// TwinCAT 3 PLC project ED_PROG
// ProgramVersion: 3.1.4026.12
// libraries:
//   Tc2_OpcUA, * (Beckhoff Automation GmbH)
//   Tc2_Standard, * (Beckhoff Automation GmbH)
//   Tc2_System, * (Beckhoff Automation GmbH)
//   Tc2_Utilities, * (Beckhoff Automation GmbH)
//   Tc3_Module, * (Beckhoff Automation GmbH)
// project tree:
//   GVLs/ opc.TcGVL, plccomms.TcGVL
//   / PlcTask.TcTTO
//   POUs/ alarm_manager.TcPOU, idle.TcPOU, cip.TcPOU, example_loop_control.TcPOU, faults.TcPOU, interlocks.TcPOU, io_mapping.TcPOU, communications.TcPOU (not stored), general.TcPOU, manual_mode.TcPOU, maint_mode.TcPOU, opc_control.TcPOU (not stored), opc_mapping.TcPOU, output_mapping.TcPOU, pump_manager.TcPOU, state_transition.TcPOU (not stored), stopping_mode.TcPOU, valve_manager.TcPOU
//   POUs/Function Blocks/ ramp.TcPOU, alarm.TcPOU, analog_scaling.TcPOU (not stored), date_time.TcPOU (not stored), motor_starter.TcPOU (not stored), motor_vfd.TcPOU (not stored), valve_analog.TcPOU (not stored), valve_digital.TcPOU (not stored)
// real-time tasks:
//   TASK PlcTask: cycle T#10ms, priority 20, ADS port 350
//   TASK twinsafe: cycle T#10ms, priority 1, ADS port 301
// I/O:
//   DEVICE Device 1 (EtherCAT), AmsNetId 10.60.1.103.2.1
//     Term 1 (EK1200) [EK1200-5000 EtherCAT Power supply (2A E-Bus)]
//       Term 2 (EL3058) [EL3058 8Ch. Ana. Input 4-20mA]
//       Term 3 (EL3058) [EL3058 8Ch. Ana. Input 4-20mA]
//       Term 4 (EL4124) [EL4124 4Ch. Ana. Output 4-20mA, 16bit]
//       Term 5 (EL4124) [EL4124 4Ch. Ana. Output 4-20mA, 16bit]
//       Term 6 (EL4124) [EL4124 4Ch. Ana. Output 4-20mA, 16bit]
//       Term 7 (EL1859) [EL1859 8Ch. Dig. Input 24V, 3ms, 8Ch. Dig. Output 24V, 0.5A]
//       Term 8 (EL1859) [EL1859 8Ch. Dig. Input 24V, 3ms, 8Ch. Dig. Output 24V, 0.5A]
//       Term 9 (EL1859) [EL1859 8Ch. Dig. Input 24V, 3ms, 8Ch. Dig. Output 24V, 0.5A]
//       Term 10 (EL1904) [EL1904, 4 Ch. Safety Input 24V, TwinSAFE]
//         modules: Module 1 (FSOES)
//       Term 11 (EL2911) [EL2911, Potential supply terminal (10 A) with 4 Ch. Safety Inputs, TwinSAFE]
//         modules: Module 2 (FSOUT), Module 3 (DEVICEIO), Module 4 (FSLOGIC)
//       Term 12 (EK1110) [EK1110 EtherCAT extension]
//     Term 20 (EK1100-0018) [EK1100-0018 EtherCAT-Koppler (2A E-Bus, erw. Surge Schutz)]
//       Term 21 (EL3058) [EL3058 8Ch. Ana. Input 4-20mA]
//       Term 22 (EL3058) [EL3058 8Ch. Ana. Input 4-20mA]
//       Term 23 (EL3058) [EL3058 8Ch. Ana. Input 4-20mA]
//       Term 24 (EL3058) [EL3058 8Ch. Ana. Input 4-20mA]
//       Term 25 (EL3058) [EL3058 8Ch. Ana. Input 4-20mA]
//       Term 26 (EL4124) [EL4124 4Ch. Ana. Output 4-20mA, 16bit]
//       Term 27 (EL4124) [EL4124 4Ch. Ana. Output 4-20mA, 16bit]
//       Term 28 (EL1859) [EL1859 8Ch. Dig. Input 24V, 3ms, 8Ch. Dig. Output 24V, 0.5A]
//       Term 29 (EL1859) [EL1859 8Ch. Dig. Input 24V, 3ms, 8Ch. Dig. Output 24V, 0.5A]
//       Term 30 (EL9011) [EL9011 End Terminal]
//     Term 31 (EK1914) [EK1914, 2 Ch. Safety Input/Output 24V,  TwinSAFE]
//       modules: Module 1 (FSOE), Module 2 (DIO)
//       Term 32 (EL1859) [EL1859 8Ch. Dig. Input 24V, 3ms, 8Ch. Dig. Output 24V, 0.5A]
//       Term 33 (EL1859) [EL1859 8Ch. Dig. Input 24V, 3ms, 8Ch. Dig. Output 24V, 0.5A]
//       Term 34 (EL1904) [EL1904, 4 Ch. Safety Input 24V, TwinSAFE]
//         modules: Module 1 (FSOES)
//       Term 35 (EL9011) [EL9011 End Terminal]
//   DEVICE Device 4 (EtherCAT), AmsNetId 10.60.1.103.5.1
//     Term 13 (EK1100-0018) [EK1100-0018 EtherCAT-Koppler (2A E-Bus, erw. Surge Schutz)]
//       Term 14 (EL3058) [EL3058 8Ch. Ana. Input 4-20mA]
//       Term 15 (EL3058) [EL3058 8Ch. Ana. Input 4-20mA]
//       Term 16 (EL3058) [EL3058 8Ch. Ana. Input 4-20mA]
//       Term 17 (EL3058) [EL3058 8Ch. Ana. Input 4-20mA]
//       Term 18 (EL3058) [EL3058 8Ch. Ana. Input 4-20mA]
//       Term 19 (EL4124) [EL4124 4Ch. Ana. Output 4-20mA, 16bit]
//       Term 20 (EL4124) [EL4124 4Ch. Ana. Output 4-20mA, 16bit]
//       Term 21 (EL1859) [EL1859 8Ch. Dig. Input 24V, 3ms, 8Ch. Dig. Output 24V, 0.5A]
//       Term 22 (EL1859) [EL1859 8Ch. Dig. Input 24V, 3ms, 8Ch. Dig. Output 24V, 0.5A]
//       Term 41 (EL9011) [EL9011 End Terminal]
//     Term 31 (EK1914) [EK1914, 2 Ch. Safety Input/Output 24V,  TwinSAFE]
//       modules: Module 1 (FSOE), Module 2 (DIO)
//       Term 32 (EL1859) [EL1859 8Ch. Dig. Input 24V, 3ms, 8Ch. Dig. Output 24V, 0.5A]
//       Term 33 (EL1859) [EL1859 8Ch. Dig. Input 24V, 3ms, 8Ch. Dig. Output 24V, 0.5A]
//       Term 34 (EL1904) [EL1904, 4 Ch. Safety Input 24V, TwinSAFE]
//         modules: Module 1 (FSOES)
//       Term 42 (EL9011) [EL9011 End Terminal]
//     Term 40 (EK1100) [EK1100 EtherCAT Coupler (2A E-Bus)]
//       Term 41 (EL3058) [EL3058 8Ch. Ana. Input 4-20mA]
//       Term 42 (EL4124) [EL4124 4Ch. Ana. Output 4-20mA, 16bit]
//       Term 43 (EL1859) [EL1859 8Ch. Dig. Input 24V, 3ms, 8Ch. Dig. Output 24V, 0.5A]
//       Term 44 (EL2911) [EL2911, Potential supply terminal (10 A) with 4 Ch. Safety Inputs, TwinSAFE]
//         modules: Module 1 (FSOE), Module 2 (FSOUT), Module 3 (DEVICEIO), Module 4 (FSLOGIC)
//       Term 43 (EL9011) [EL9011 End Terminal]
// variable links:
//   Device 1 (EtherCAT) <-> Device 1 (EtherCAT)/Term 1 (EK1200)/Term 11 (EL2911)
//     Term 31 (EK1914)/Module 1 (FSOE)/Inputs/FSOE <-> ConnectionOutputs/Message_18 RxPDO
//     Term 31 (EK1914)/Module 1 (FSOE)/Outputs/FSOE <-> ConnectionInputs/Message_18 TxPDO
//   ED2_PROG Instance <-> Device 1 (EtherCAT)/Term 1 (EK1200)/Term 2 (EL3058)
//     PlcTask Inputs/io_mapping.u_3112_b_speed_feedback_raw_input <-> AI Standard Channel 1/Value
//     PlcTask Inputs/io_mapping.u_3160_b_speed_feedback_raw_input <-> AI Standard Channel 4/Value
//     PlcTask Inputs/io_mapping.u_3212_b_speed_feedback_raw_input <-> AI Standard Channel 2/Value
//     PlcTask Inputs/io_mapping.u_3260_b_speed_feedback_raw_input <-> AI Standard Channel 5/Value
//     PlcTask Inputs/io_mapping.u_3312_b_speed_feedback_raw_input <-> AI Standard Channel 3/Value
//     PlcTask Inputs/io_mapping.u_3360_b_speed_feedback_raw_input <-> AI Standard Channel 6/Value
//     PlcTask Inputs/io_mapping.u_3370_b_speed_feedback_raw_input <-> AI Standard Channel 7/Value
//   ED2_PROG Instance <-> Device 1 (EtherCAT)/Term 1 (EK1200)/Term 4 (EL4124)
//     PlcTask Outputs/output_mapping.u_3112_b_speed_command_io <-> AO Output Channel 1/Analog output
//     PlcTask Outputs/output_mapping.u_3160_b_speed_command_io <-> AO Output Channel 4/Analog output
//     PlcTask Outputs/output_mapping.u_3212_b_speed_command_io <-> AO Output Channel 2/Analog output
//     PlcTask Outputs/output_mapping.u_3312_b_speed_command_io <-> AO Output Channel 3/Analog output
//   ED2_PROG Instance <-> Device 1 (EtherCAT)/Term 1 (EK1200)/Term 5 (EL4124)
//     PlcTask Outputs/output_mapping.u_3260_b_speed_command_io <-> AO Output Channel 1/Analog output
//     PlcTask Outputs/output_mapping.u_3360_b_speed_command_io <-> AO Output Channel 2/Analog output
//     PlcTask Outputs/output_mapping.u_3370_b_speed_command_io <-> AO Output Channel 3/Analog output
//   ED2_PROG Instance <-> Device 1 (EtherCAT)/Term 1 (EK1200)/Term 7 (EL1859)
//     PlcTask Inputs/io_mapping.u_3112_b_fault_feedback <-> Channel 1/Input
//     PlcTask Inputs/io_mapping.u_3160_b_fault_feedback <-> Channel 7/Input
//     PlcTask Inputs/io_mapping.u_3212_b_fault_feedback <-> Channel 3/Input
//     PlcTask Inputs/io_mapping.u_3312_b_fault_feedback <-> Channel 5/Input
//     PlcTask Inputs/io_mapping.u_3112_b_run_feedback <-> Channel 2/Input
//     PlcTask Inputs/io_mapping.u_3160_b_run_feedback <-> Channel 8/Input
//     PlcTask Inputs/io_mapping.u_3212_b_run_feedback <-> Channel 4/Input
//     PlcTask Inputs/io_mapping.u_3312_b_run_feedback <-> Channel 6/Input
//     PlcTask Outputs/output_mapping.u_3112_b_fault_reset_io <-> Channel 10/Output
//     PlcTask Outputs/output_mapping.u_3160_b_fault_reset_io <-> Channel 16/Output
//     PlcTask Outputs/output_mapping.u_3212_b_fault_reset_io <-> Channel 12/Output
//     PlcTask Outputs/output_mapping.u_3312_b_fault_reset_io <-> Channel 14/Output
//     PlcTask Outputs/output_mapping.u_3112_b_run_command_io <-> Channel 9/Output
//     PlcTask Outputs/output_mapping.u_3160_b_run_command_io <-> Channel 15/Output
//     PlcTask Outputs/output_mapping.u_3212_b_run_command_io <-> Channel 11/Output
//     PlcTask Outputs/output_mapping.u_3312_b_run_command_io <-> Channel 13/Output
//   ED2_PROG Instance <-> Device 1 (EtherCAT)/Term 1 (EK1200)/Term 8 (EL1859)
//     PlcTask Inputs/io_mapping.u_3260_b_fault_feedback <-> Channel 1/Input
//     PlcTask Inputs/io_mapping.u_3360_b_fault_feedback <-> Channel 3/Input
//     PlcTask Inputs/io_mapping.u_3370_b_fault_feedback <-> Channel 5/Input
//     PlcTask Inputs/io_mapping.u_3260_b_run_feedback <-> Channel 2/Input
//     PlcTask Inputs/io_mapping.u_3360_b_run_feedback <-> Channel 4/Input
//     PlcTask Inputs/io_mapping.u_3370_b_run_feedback <-> Channel 6/Input
//     PlcTask Outputs/output_mapping.u_3260_b_fault_reset_io <-> Channel 10/Output
//     PlcTask Outputs/output_mapping.u_3360_b_fault_reset_io <-> Channel 12/Output
//     PlcTask Outputs/output_mapping.u_3370_b_fault_reset_io <-> Channel 14/Output
//     PlcTask Outputs/output_mapping.u_3260_b_run_command_io <-> Channel 9/Output
//     PlcTask Outputs/output_mapping.u_3360_b_run_command_io <-> Channel 11/Output
//     PlcTask Outputs/output_mapping.u_3370_b_run_command_io <-> Channel 13/Output
//   ED2_PROG Instance <-> Device 1 (EtherCAT)/Term 20 (EK1100-0018)/Term 21 (EL3058)
//     PlcTask Inputs/io_mapping.pt_3119_b_raw_input <-> AI Standard Channel 1/Value
//     PlcTask Inputs/io_mapping.pt_3141_b_raw_input <-> AI Standard Channel 4/Value
//     PlcTask Inputs/io_mapping.pt_3219_b_raw_input <-> AI Standard Channel 2/Value
//     PlcTask Inputs/io_mapping.pt_3241_b_raw_input <-> AI Standard Channel 5/Value
//     PlcTask Inputs/io_mapping.pt_3319_b_raw_input <-> AI Standard Channel 3/Value
//     PlcTask Inputs/io_mapping.pt_3341_b_raw_input <-> AI Standard Channel 6/Value
//     PlcTask Inputs/io_mapping.tt_3118_b_raw_input <-> AI Standard Channel 7/Value
//     PlcTask Inputs/io_mapping.tt_3218_b_raw_input <-> AI Standard Channel 8/Value
//   ED2_PROG Instance <-> Device 1 (EtherCAT)/Term 20 (EK1100-0018)/Term 22 (EL3058)
//     PlcTask Inputs/io_mapping.av_3148_b_position_feedback_raw_input <-> AI Standard Channel 8/Value
//     PlcTask Inputs/io_mapping.tt_3140_b_raw_input <-> AI Standard Channel 2/Value
//     PlcTask Inputs/io_mapping.tt_3240_b_raw_input <-> AI Standard Channel 3/Value
//     PlcTask Inputs/io_mapping.tt_3318_b_raw_input <-> AI Standard Channel 1/Value
//     PlcTask Inputs/io_mapping.tt_3340_b_raw_input <-> AI Standard Channel 4/Value
//   ED2_PROG Instance <-> Device 1 (EtherCAT)/Term 20 (EK1100-0018)/Term 23 (EL3058)
//     PlcTask Inputs/io_mapping.av_3248_b_position_feedback_raw_input <-> AI Standard Channel 1/Value
//     PlcTask Inputs/io_mapping.av_3348_b_position_feedback_raw_input <-> AI Standard Channel 2/Value
//     PlcTask Inputs/io_mapping.lt_3102_b_raw_input <-> AI Standard Channel 3/Value
//     PlcTask Inputs/io_mapping.lt_3153_b_raw_input <-> AI Standard Channel 6/Value
//     PlcTask Inputs/io_mapping.lt_3202_b_raw_input <-> AI Standard Channel 4/Value
//     PlcTask Inputs/io_mapping.lt_3253_b_raw_input <-> AI Standard Channel 7/Value
//     PlcTask Inputs/io_mapping.lt_3302_b_raw_input <-> AI Standard Channel 5/Value
//     PlcTask Inputs/io_mapping.lt_3353_b_raw_input <-> AI Standard Channel 8/Value
//   ED2_PROG Instance <-> Device 1 (EtherCAT)/Term 20 (EK1100-0018)/Term 24 (EL3058)
//     PlcTask Inputs/io_mapping.cct_3120_b_raw_input <-> AI Standard Channel 1/Value
//     PlcTask Inputs/io_mapping.cct_3142_b_raw_input <-> AI Standard Channel 4/Value
//     PlcTask Inputs/io_mapping.cct_3220_b_raw_input <-> AI Standard Channel 2/Value
//     PlcTask Inputs/io_mapping.cct_3242_b_raw_input <-> AI Standard Channel 5/Value
//     PlcTask Inputs/io_mapping.cct_3320_b_raw_input <-> AI Standard Channel 3/Value
//     PlcTask Inputs/io_mapping.cct_3342_b_raw_input <-> AI Standard Channel 6/Value
//   ED2_PROG Instance <-> Device 1 (EtherCAT)/Term 20 (EK1100-0018)/Term 25 (EL3058)
//     PlcTask Inputs/io_mapping.ft_3122_b_raw_input <-> AI Standard Channel 1/Value
//     PlcTask Inputs/io_mapping.ft_3222_b_raw_input <-> AI Standard Channel 2/Value
//     PlcTask Inputs/io_mapping.ft_3322_b_raw_input <-> AI Standard Channel 3/Value
//   ED2_PROG Instance <-> Device 1 (EtherCAT)/Term 20 (EK1100-0018)/Term 26 (EL4124)
//     PlcTask Outputs/output_mapping.av_3148_b_position_command_io <-> AO Output Channel 1/Analog output
//     PlcTask Outputs/output_mapping.av_3248_b_position_command_io <-> AO Output Channel 2/Analog output
//     PlcTask Outputs/output_mapping.av_3348_b_position_command_io <-> AO Output Channel 3/Analog output
//   ED2_PROG Instance <-> Device 1 (EtherCAT)/Term 20 (EK1100-0018)/Term 28 (EL1859)
//     PlcTask Inputs/io_mapping.nv_3135_b_open_feedback <-> Channel 1/Input
//     PlcTask Inputs/io_mapping.nv_3162_b_open_feedback <-> Channel 5/Input
//     PlcTask Inputs/io_mapping.nv_3235_b_open_feedback <-> Channel 2/Input
//     PlcTask Inputs/io_mapping.nv_3335_b_open_feedback <-> Channel 3/Input
//     PlcTask Inputs/io_mapping.nv_3372_b_open_feedback <-> Channel 4/Input
//   ED2_PROG Instance <-> Device 1 (EtherCAT)/Term 20 (EK1100-0018)/Term 29 (EL1859)
//     PlcTask Inputs/io_mapping.nv_3135_b_closed_feedback <-> Channel 1/Input
//     PlcTask Inputs/io_mapping.nv_3162_b_closed_feedback <-> Channel 5/Input
//     PlcTask Inputs/io_mapping.nv_3235_b_closed_feedback <-> Channel 2/Input
//     PlcTask Inputs/io_mapping.nv_3335_b_closed_feedback <-> Channel 3/Input
//     PlcTask Inputs/io_mapping.nv_3372_b_closed_feedback <-> Channel 4/Input
//   ED2_PROG Instance <-> Device 1 (EtherCAT)/Term 31 (EK1914)/Term 32 (EL1859)
//     PlcTask Outputs/output_mapping.nv_3110_b_open_command_io <-> Channel 11/Output
//     PlcTask Outputs/output_mapping.nv_3135_b_open_command_io <-> Channel 12/Output
//     PlcTask Outputs/output_mapping.nv_3162_b_open_command_io <-> Channel 9/Output
//     PlcTask Outputs/output_mapping.nv_3210_b_open_command_io <-> Channel 10/Output
//     PlcTask Outputs/output_mapping.nv_3235_b_open_command_io <-> Channel 14/Output
//     PlcTask Outputs/output_mapping.nv_3310_b_open_command_io <-> Channel 13/Output
//     PlcTask Outputs/output_mapping.nv_3335_b_open_command_io <-> Channel 15/Output
//     PlcTask Outputs/output_mapping.nv_3372_b_open_command_io <-> Channel 16/Output

CONFIGURATION ED_PROG
    RESOURCE PLC ON TwinCAT3
        TASK PlcTask(INTERVAL := T#10ms, PRIORITY := 20);
        PROGRAM communications WITH PlcTask : communications;
        PROGRAM example_loop_control WITH PlcTask : example_loop_control;
        PROGRAM general WITH PlcTask : general;
        PROGRAM interlocks WITH PlcTask : interlocks;
        PROGRAM io_mapping WITH PlcTask : io_mapping;
        PROGRAM opc_control WITH PlcTask : opc_control;
        PROGRAM opc_mapping WITH PlcTask : opc_mapping;
        PROGRAM state_transition WITH PlcTask : state_transition;
        PROGRAM manual_mode WITH PlcTask : manual_mode;
        PROGRAM valve_manager WITH PlcTask : valve_manager;
        PROGRAM stopping_mode WITH PlcTask : stopping_mode;
        PROGRAM pump_manager WITH PlcTask : pump_manager;
        PROGRAM idle WITH PlcTask : idle;
        PROGRAM maint_mode WITH PlcTask : maint_mode;
        PROGRAM faults WITH PlcTask : faults;
        PROGRAM alarm_manager WITH PlcTask : alarm_manager;
        PROGRAM cip WITH PlcTask : cip;
    END_RESOURCE
END_CONFIGURATION

// ---- GVLs/opc.TcGVL
{attribute 'qualified_only'}
{attribute 'global_init_slot' := '50500'}
VAR_GLOBAL PERSISTENT
	//These tags are created here because you cannot write directly to local scoped tags(cpt_3144) from outside the POU
	//They are created here then mapped to the local variables in the POU
	//All tags in this GVL MUST have the {attribute 'OPC.UA.DA' :='1'} string above them in order to be exposed to OPC
	//Tags that are ONLY being read from the HMI have their values set in the opc_mapping program
	
	//------------------------------------------------------------------------------------------------------------------


	//---System date time year-----------------------------------------------------------------------------------------------
	{attribute 'OPC.UA.DA' :='1'}
	popa_0081_system_date_time_year : INT;
	//System date time month
	{attribute 'OPC.UA.DA' :='1'}
	popa_0081_system_date_time_month : INT;
	//System date time day
	{attribute 'OPC.UA.DA' :='1'}
	popa_0081_system_date_time_day : INT;
	//System date time hour
	{attribute 'OPC.UA.DA' :='1'}
	popa_0081_system_date_time_hour : INT;
	//System date time minute
	{attribute 'OPC.UA.DA' :='1'}
	popa_0081_system_date_time_minute : INT;
	//System date time second
	{attribute 'OPC.UA.DA' :='1'}
	popa_0081_system_date_time_second : INT;
	//Hour setpoint for daily reset triggers
	{attribute 'OPC.UA.DA' :='1'}
	popa_0081_daily_reset_hour_setpoint : INT;
	//Minute setpoint for daily reset triggers
	{attribute 'OPC.UA.DA' :='1'}
	popa_0081_daily_reset_minute_setpoint : INT;
	//Alarm acknowledge, acks all alarms, clears lower priority level alarms
	{attribute 'OPC.UA.DA' :='1'}
	popa_0081_alarm_ack : BOOL;
	//Alarm reset, clears higher priority alarms
	{attribute 'OPC.UA.DA' :='1'}
	popa_0081_alarm_reset : BOOL;
	
//----------------------------------------------------------------------------------------------------------------------------------------		
	//State Mode
	{attribute 'OPC.UA.DA' :='1'}
	popa_0081_ed_routine_maint : BOOL;
	{attribute 'OPC.UA.DA' :='1'}
	popa_0081_ed_routine_idle : BOOL;
	{attribute 'OPC.UA.DA' :='1'}
	popa_0081_ed_routine_cip : BOOL;
	{attribute 'OPC.UA.DA' :='1'}
	popa_0081_ed_routine_stop : BOOL;
	{attribute 'OPC.UA.DA' :='1'}
	popa_0081_ed_routine_critical_stop : BOOL;
	
	
	//Safety
	{attribute 'OPC.UA.DA' :='1'}
	popa_0081_ed_safety_reset : BOOL;
	
	
//---HMI Commands--------------------------------------------------------------------------------------------------------------------------------------

	//Setpoints------------------------------------------------------------------------------------------------------------------
	{attribute 'OPC.UA.DA' :='1'}
	popa_0081_idle_pressure_setpoint_request : REAL;
	{attribute 'OPC.UA.DA' :='1'}
	popa_0081_cip_pressure_setpoint_request : REAL;
	{attribute 'OPC.UA.DA' :='1'}
	popa_0081_av_3148_a_hmi_position_request : REAL;
	{attribute 'OPC.UA.DA' :='1'}
	popa_0081_av_3248_a_hmi_position_request : REAL;
	{attribute 'OPC.UA.DA' :='1'}
	popa_0081_av_3348_a_hmi_position_request : REAL;
	
	//Pumps-----------------------------------------------------------------------------------------------------------------------
	{attribute 'OPC.UA.DA' :='1'}
	popa_0081_u_3112_a_hmi_start_request: BOOL;
	{attribute 'OPC.UA.DA' :='1'}
	popa_0081_u_3212_a_hmi_start_request: BOOL;
	{attribute 'OPC.UA.DA' :='1'}
	popa_0081_u_3312_a_hmi_start_request: BOOL;
	{attribute 'OPC.UA.DA' :='1'}
	popa_0081_u_3160_a_hmi_start_request: BOOL;
	{attribute 'OPC.UA.DA' :='1'}
	popa_0081_u_3260_a_hmi_start_request: BOOL;
	{attribute 'OPC.UA.DA' :='1'}
	popa_0081_u_3360_a_hmi_start_request: BOOL;
	{attribute 'OPC.UA.DA' :='1'}
	popa_0081_u_3370_a_hmi_start_request: BOOL;
	{attribute 'OPC.UA.DA' :='1'}
	popa_0091_u_3405_a_hmi_start_request: BOOL;
		
	{attribute 'OPC.UA.DA' :='1'}
	popa_0081_u_3112_a_hmi_speed_request: REAL;
	{attribute 'OPC.UA.DA' :='1'}
	popa_0081_u_3212_a_hmi_speed_request: REAL;
	{attribute 'OPC.UA.DA' :='1'}
	popa_0081_u_3312_a_hmi_speed_request: REAL;
	{attribute 'OPC.UA.DA' :='1'}
	popa_0081_u_3160_a_hmi_speed_request: REAL;
	{attribute 'OPC.UA.DA' :='1'}
	popa_0081_u_3260_a_hmi_speed_request: REAL;
	{attribute 'OPC.UA.DA' :='1'}
	popa_0081_u_3360_a_hmi_speed_request: REAL;
	{attribute 'OPC.UA.DA' :='1'}
	popa_0081_u_3370_a_hmi_speed_request: REAL;
	{attribute 'OPC.UA.DA' :='1'}
	popa_0091_u_3405_a_hmi_speed_request: REAL;
	
	//Valves------------------------------------------------------------------------------------------------------------------------------
	{attribute 'OPC.UA.DA' :='1'}
	popa_0081_nv_3110_a_hmi_open_request: BOOL;
	{attribute 'OPC.UA.DA' :='1'}
	popa_0081_nv_3210_a_hmi_open_request: BOOL;
	{attribute 'OPC.UA.DA' :='1'}
	popa_0081_nv_3310_a_hmi_open_request: BOOL;
	{attribute 'OPC.UA.DA' :='1'}
	popa_0081_nv_3135_a_hmi_open_request: BOOL;
	{attribute 'OPC.UA.DA' :='1'}
	popa_0081_nv_3235_a_hmi_open_request: BOOL;
	{attribute 'OPC.UA.DA' :='1'}
	popa_0081_nv_3335_a_hmi_open_request: BOOL;
	{attribute 'OPC.UA.DA' :='1'}
	popa_0081_nv_3372_a_hmi_open_request: BOOL;
	{attribute 'OPC.UA.DA' :='1'}
	popa_0081_nv_3162_a_hmi_open_request: BOOL;
	

	//-------------------------------------------------------------------------------------------
	//Digital valve open request
	{attribute 'OPC.UA.DA' :='1'}
	popa_0081_nv_3110_a_open_request : BOOL;
	//Digital valve status
	{attribute 'OPC.UA.DA' :='1'}
	popa_0081_nv_3110_a_status : INT;
	
	//Digital valve open request
	{attribute 'OPC.UA.DA' :='1'}
	popa_0081_nv_3210_a_open_request : BOOL;
	//Digital valve status
	{attribute 'OPC.UA.DA' :='1'}
	popa_0081_nv_3210_a_status : INT;
	
	//Digital valve open request
	{attribute 'OPC.UA.DA' :='1'}
	popa_0081_nv_3310_a_open_request : BOOL;
	//Digital valve status
	{attribute 'OPC.UA.DA' :='1'}
	popa_0081_nv_3310_a_status : INT;
	
	//Digital valve open request
	{attribute 'OPC.UA.DA' :='1'}
	popa_0081_nv_3135_a_open_request : BOOL;
	//Digital valve status
	{attribute 'OPC.UA.DA' :='1'}
	popa_0081_nv_3135_a_status : INT;
	
	//Digital valve open request
	{attribute 'OPC.UA.DA' :='1'}
	popa_0081_nv_3235_a_open_request : BOOL;
	//Digital valve status
	{attribute 'OPC.UA.DA' :='1'}
	popa_0081_nv_3235_a_status : INT;
	
	//Digital valve open request
	{attribute 'OPC.UA.DA' :='1'}
	popa_0081_nv_3335_a_open_request : BOOL;
	//Digital valve status
	{attribute 'OPC.UA.DA' :='1'}
	popa_0081_nv_3335_a_status : INT;
	
	//Digital valve open request
	{attribute 'OPC.UA.DA' :='1'}
	popa_0081_nv_3372_a_open_request : BOOL;
	//Digital valve status
	{attribute 'OPC.UA.DA' :='1'}
	popa_0081_nv_3372_a_status : INT;
	
	//Digital valve open request
	{attribute 'OPC.UA.DA' :='1'}
	popa_0081_nv_3162_a_open_request : BOOL;
	//Digital valve status
	{attribute 'OPC.UA.DA' :='1'}
	popa_0081_nv_3162_a_status : INT;
	
	//------------------------------------------------------------------------------------------------------------------
	//Alarm Priority setpoint
	{attribute 'OPC.UA.DA' :='1'}
	popa_0081_av_3148_a_position_fail_priority : INT;
	//Alarm delay setpoint(seconds)
	{attribute 'OPC.UA.DA' :='1'}
	popa_0081_av_3148_a_position_fail_delay_setpoint : INT;
	//Alarm active for HMI
	{attribute 'OPC.UA.DA' :='1'}
	popa_0081_av_3148_a_position_fail_active : BOOL;
	//Alarm enable
	{attribute 'OPC.UA.DA' :='1'}
	popa_0081_av_3148_a_position_fail_enable: BOOL;
	//------------------------------------------------------------------------------------------------------------------
	//Alarm Priority setpoint
	{attribute 'OPC.UA.DA' :='1'}
	popa_0081_av_3248_a_position_fail_priority : INT;
	//Alarm delay setpoint(seconds)
	{attribute 'OPC.UA.DA' :='1'}
	popa_0081_av_3248_a_position_fail_delay_setpoint : INT;
	//Alarm active for HMI
	{attribute 'OPC.UA.DA' :='1'}
	popa_0081_av_3248_a_position_fail_active : BOOL;
	//Alarm enable
	{attribute 'OPC.UA.DA' :='1'}
	popa_0081_av_3248_a_position_fail_enable: BOOL;
	//------------------------------------------------------------------------------------------------------------------
	//Alarm Priority setpoint
	{attribute 'OPC.UA.DA' :='1'}
	popa_0081_av_3348_a_position_fail_priority : INT;
	//Alarm delay setpoint(seconds)
	{attribute 'OPC.UA.DA' :='1'}
	popa_0081_av_3348_a_position_fail_delay_setpoint : INT;
	//Alarm active for HMI
	{attribute 'OPC.UA.DA' :='1'}
	popa_0081_av_3348_a_position_fail_active : BOOL;
	//Alarm enable
	{attribute 'OPC.UA.DA' :='1'}
	popa_0081_av_3348_a_position_fail_enable: BOOL;
	
	//------------------------------------------------------------------------------------------------------------------
	//Alarm Priority setpoint
	{attribute 'OPC.UA.DA' :='1'}
	popa_0081_nv_3110_a_fail_to_open_priority : INT;
	//Alarm delay setpoint(seconds)
	{attribute 'OPC.UA.DA' :='1'}
	popa_0081_nv_3110_a_fail_to_open_delay_setpoint : INT;
	//Alarm active for HMI
	{attribute 'OPC.UA.DA' :='1'}
	popa_0081_nv_3110_a_fail_to_open_active : BOOL;
	//Alarm enable
	{attribute 'OPC.UA.DA' :='1'}
	popa_0081_nv_3110_a_fail_to_open_enable: BOOL;
	
	//Alarm Priority setpoint
	{attribute 'OPC.UA.DA' :='1'}
	popa_0081_nv_3110_a_fail_to_close_priority : INT;
	//Alarm delay setpoint(seconds)
	{attribute 'OPC.UA.DA' :='1'}
	popa_0081_nv_3110_a_fail_to_close_delay_setpoint : INT;
	//Alarm active for HMI
	{attribute 'OPC.UA.DA' :='1'}
	popa_0081_nv_3110_a_fail_to_close_active : BOOL;
	//Alarm enable
	{attribute 'OPC.UA.DA' :='1'}
	popa_0081_nv_3110_a_fail_to_close_enable: BOOL;
	
	//------------------------------------------------------------------------------------------------------------------
	//Alarm Priority setpoint
	{attribute 'OPC.UA.DA' :='1'}
	popa_0081_nv_3210_a_fail_to_open_priority : INT;
	//Alarm delay setpoint(seconds)
	{attribute 'OPC.UA.DA' :='1'}
	popa_0081_nv_3210_a_fail_to_open_delay_setpoint : INT;
	//Alarm active for HMI
	{attribute 'OPC.UA.DA' :='1'}
	popa_0081_nv_3210_a_fail_to_open_active : BOOL;
	//Alarm enable
	{attribute 'OPC.UA.DA' :='1'}
	popa_0081_nv_3210_a_fail_to_open_enable: BOOL;
	
	//Alarm Priority setpoint
	{attribute 'OPC.UA.DA' :='1'}
	popa_0081_nv_3210_a_fail_to_close_priority : INT;
	//Alarm delay setpoint(seconds)
	{attribute 'OPC.UA.DA' :='1'}
	popa_0081_nv_3210_a_fail_to_close_delay_setpoint : INT;
	//Alarm active for HMI
	{attribute 'OPC.UA.DA' :='1'}
	popa_0081_nv_3210_a_fail_to_close_active : BOOL;
	//Alarm enable
	{attribute 'OPC.UA.DA' :='1'}
	popa_0081_nv_3210_a_fail_to_close_enable: BOOL;
	
	//------------------------------------------------------------------------------------------------------------------
	//Alarm Priority setpoint
	{attribute 'OPC.UA.DA' :='1'}
	popa_0081_nv_3310_a_fail_to_open_priority : INT;
	//Alarm delay setpoint(seconds)
	{attribute 'OPC.UA.DA' :='1'}
	popa_0081_nv_3310_a_fail_to_open_delay_setpoint : INT;
	//Alarm active for HMI
	{attribute 'OPC.UA.DA' :='1'}
	popa_0081_nv_3310_a_fail_to_open_active : BOOL;
	//Alarm enable
	{attribute 'OPC.UA.DA' :='1'}
	popa_0081_nv_3310_a_fail_to_open_enable: BOOL;
	
	//Alarm Priority setpoint
	{attribute 'OPC.UA.DA' :='1'}
	popa_0081_nv_3310_a_fail_to_close_priority : INT;
	//Alarm delay setpoint(seconds)
	{attribute 'OPC.UA.DA' :='1'}
	popa_0081_nv_3310_a_fail_to_close_delay_setpoint : INT;
	//Alarm active for HMI
	{attribute 'OPC.UA.DA' :='1'}
	popa_0081_nv_3310_a_fail_to_close_active : BOOL;
	//Alarm enable
	{attribute 'OPC.UA.DA' :='1'}
	popa_0081_nv_3310_a_fail_to_close_enable: BOOL;
	
	//------------------------------------------------------------------------------------------------------------------
	//Alarm Priority setpoint
	{attribute 'OPC.UA.DA' :='1'}
	popa_0081_nv_3135_a_fail_to_open_priority : INT;
	//Alarm delay setpoint(seconds)
	{attribute 'OPC.UA.DA' :='1'}
	popa_0081_nv_3135_a_fail_to_open_delay_setpoint : INT;
	//Alarm active for HMI
	{attribute 'OPC.UA.DA' :='1'}
	popa_0081_nv_3135_a_fail_to_open_active : BOOL;
	//Alarm enable
	{attribute 'OPC.UA.DA' :='1'}
	popa_0081_nv_3135_a_fail_to_open_enable: BOOL;
	
	//Alarm Priority setpoint
	{attribute 'OPC.UA.DA' :='1'}
	popa_0081_nv_3135_a_fail_to_close_priority : INT;
	//Alarm delay setpoint(seconds)
	{attribute 'OPC.UA.DA' :='1'}
	popa_0081_nv_3135_a_fail_to_close_delay_setpoint : INT;
	//Alarm active for HMI
	{attribute 'OPC.UA.DA' :='1'}
	popa_0081_nv_3135_a_fail_to_close_active : BOOL;
	//Alarm enable
	{attribute 'OPC.UA.DA' :='1'}
	popa_0081_nv_3135_a_fail_to_close_enable: BOOL;
	
	//------------------------------------------------------------------------------------------------------------------
	//Alarm Priority setpoint
	{attribute 'OPC.UA.DA' :='1'}
	popa_0081_nv_3235_a_fail_to_open_priority : INT;
	//Alarm delay setpoint(seconds)
	{attribute 'OPC.UA.DA' :='1'}
	popa_0081_nv_3235_a_fail_to_open_delay_setpoint : INT;
	//Alarm active for HMI
	{attribute 'OPC.UA.DA' :='1'}
	popa_0081_nv_3235_a_fail_to_open_active : BOOL;
	//Alarm enable
	{attribute 'OPC.UA.DA' :='1'}
	popa_0081_nv_3235_a_fail_to_open_enable: BOOL;
	
	//Alarm Priority setpoint
	{attribute 'OPC.UA.DA' :='1'}
	popa_0081_nv_3235_a_fail_to_close_priority : INT;
	//Alarm delay setpoint(seconds)
	{attribute 'OPC.UA.DA' :='1'}
	popa_0081_nv_3235_a_fail_to_close_delay_setpoint : INT;
	//Alarm active for HMI
	{attribute 'OPC.UA.DA' :='1'}
	popa_0081_nv_3235_a_fail_to_close_active : BOOL;
	//Alarm enable
	{attribute 'OPC.UA.DA' :='1'}
	popa_0081_nv_3235_a_fail_to_close_enable: BOOL;
	
	//------------------------------------------------------------------------------------------------------------------
	//Alarm Priority setpoint
	{attribute 'OPC.UA.DA' :='1'}
	popa_0081_nv_3335_a_fail_to_open_priority : INT;
	//Alarm delay setpoint(seconds)
	{attribute 'OPC.UA.DA' :='1'}
	popa_0081_nv_3335_a_fail_to_open_delay_setpoint : INT;
	//Alarm active for HMI
	{attribute 'OPC.UA.DA' :='1'}
	popa_0081_nv_3335_a_fail_to_open_active : BOOL;
	//Alarm enable
	{attribute 'OPC.UA.DA' :='1'}
	popa_0081_nv_3335_a_fail_to_open_enable: BOOL;
	
	//Alarm Priority setpoint
	{attribute 'OPC.UA.DA' :='1'}
	popa_0081_nv_3335_a_fail_to_close_priority : INT;
	//Alarm delay setpoint(seconds)
	{attribute 'OPC.UA.DA' :='1'}
	popa_0081_nv_3335_a_fail_to_close_delay_setpoint : INT;
	//Alarm active for HMI
	{attribute 'OPC.UA.DA' :='1'}
	popa_0081_nv_3335_a_fail_to_close_active : BOOL;
	//Alarm enable
	{attribute 'OPC.UA.DA' :='1'}
	popa_0081_nv_3335_a_fail_to_close_enable: BOOL;
	
	//------------------------------------------------------------------------------------------------------------------
	//Alarm Priority setpoint
	{attribute 'OPC.UA.DA' :='1'}
	popa_0081_nv_3372_a_fail_to_open_priority : INT;
	//Alarm delay setpoint(seconds)
	{attribute 'OPC.UA.DA' :='1'}
	popa_0081_nv_3372_a_fail_to_open_delay_setpoint : INT;
	//Alarm active for HMI
	{attribute 'OPC.UA.DA' :='1'}
	popa_0081_nv_3372_a_fail_to_open_active : BOOL;
	//Alarm enable
	{attribute 'OPC.UA.DA' :='1'}
	popa_0081_nv_3372_a_fail_to_open_enable: BOOL;
	
	//Alarm Priority setpoint
	{attribute 'OPC.UA.DA' :='1'}
	popa_0081_nv_3372_a_fail_to_close_priority : INT;
	//Alarm delay setpoint(seconds)
	{attribute 'OPC.UA.DA' :='1'}
	popa_0081_nv_3372_a_fail_to_close_delay_setpoint : INT;
	//Alarm active for HMI
	{attribute 'OPC.UA.DA' :='1'}
	popa_0081_nv_3372_a_fail_to_close_active : BOOL;
	//Alarm enable
	{attribute 'OPC.UA.DA' :='1'}
	popa_0081_nv_3372_a_fail_to_close_enable: BOOL;
	
	//------------------------------------------------------------------------------------------------------------------
	//Alarm Priority setpoint
	{attribute 'OPC.UA.DA' :='1'}
	popa_0081_nv_3162_a_fail_to_open_priority : INT;
	//Alarm delay setpoint(seconds)
	{attribute 'OPC.UA.DA' :='1'}
	popa_0081_nv_3162_a_fail_to_open_delay_setpoint : INT;
	//Alarm active for HMI
	{attribute 'OPC.UA.DA' :='1'}
	popa_0081_nv_3162_a_fail_to_open_active : BOOL;
	//Alarm enable
	{attribute 'OPC.UA.DA' :='1'}
	popa_0081_nv_3162_a_fail_to_open_enable: BOOL;
	
	//Alarm Priority setpoint
	{attribute 'OPC.UA.DA' :='1'}
	popa_0081_nv_3162_a_fail_to_close_priority : INT;
	//Alarm delay setpoint(seconds)
	{attribute 'OPC.UA.DA' :='1'}
	popa_0081_nv_3162_a_fail_to_close_delay_setpoint : INT;
	//Alarm active for HMI
	{attribute 'OPC.UA.DA' :='1'}
	popa_0081_nv_3162_a_fail_to_close_active : BOOL;
	//Alarm enable
	{attribute 'OPC.UA.DA' :='1'}
	popa_0081_nv_3162_a_fail_to_close_enable: BOOL;
	


//---Pumps-------------------------------------------------------------------------------------------------------------------------------------
	//------------------------------------------------------------------------------------------------------------------
	//Alarm Priority setpoint
	{attribute 'OPC.UA.DA' :='1'}
	popa_0081_u_3112_a_fail_to_start_priority : INT;
	//Alarm delay setpoint(seconds)
	{attribute 'OPC.UA.DA' :='1'}
	popa_0081_u_3112_a_fail_to_start_delay_setpoint : INT;
	//Alarm active for HMI
	{attribute 'OPC.UA.DA' :='1'}
	popa_0081_u_3112_a_fail_to_start_active : BOOL;
	//Alarm enable
	{attribute 'OPC.UA.DA' :='1'}
	popa_0081_u_3112_a_fail_to_start_enable: BOOL;
	
	//Alarm Priority setpoint
	{attribute 'OPC.UA.DA' :='1'}
	popa_0081_u_3112_a_fail_to_stop_priority : INT;
	//Alarm delay setpoint(seconds)
	{attribute 'OPC.UA.DA' :='1'}
	popa_0081_u_3112_a_fail_to_stop_delay_setpoint : INT;
	//Alarm active for HMI
	{attribute 'OPC.UA.DA' :='1'}
	popa_0081_u_3112_a_fail_to_stop_active : BOOL;
	//Alarm enable
	{attribute 'OPC.UA.DA' :='1'}
	popa_0081_u_3112_a_fail_to_stop_enable: BOOL;
	
	//------------------------------------------------------------------------------------------------------------------
	//Alarm Priority setpoint
	{attribute 'OPC.UA.DA' :='1'}
	popa_0081_u_3212_a_fail_to_start_priority : INT;
	//Alarm delay setpoint(seconds)
	{attribute 'OPC.UA.DA' :='1'}
	popa_0081_u_3212_a_fail_to_start_delay_setpoint : INT;
	//Alarm active for HMI
	{attribute 'OPC.UA.DA' :='1'}
	popa_0081_u_3212_a_fail_to_start_active : BOOL;
	//Alarm enable
	{attribute 'OPC.UA.DA' :='1'}
	popa_0081_u_3212_a_fail_to_start_enable: BOOL;
	
	//Alarm Priority setpoint
	{attribute 'OPC.UA.DA' :='1'}
	popa_0081_u_3212_a_fail_to_stop_priority : INT;
	//Alarm delay setpoint(seconds)
	{attribute 'OPC.UA.DA' :='1'}
	popa_0081_u_3212_a_fail_to_stop_delay_setpoint : INT;
	//Alarm active for HMI
	{attribute 'OPC.UA.DA' :='1'}
	popa_0081_u_3212_a_fail_to_stop_active : BOOL;
	//Alarm enable
	{attribute 'OPC.UA.DA' :='1'}
	popa_0081_u_3212_a_fail_to_stop_enable: BOOL;
	
	//------------------------------------------------------------------------------------------------------------------
	//Alarm Priority setpoint
	{attribute 'OPC.UA.DA' :='1'}
	popa_0081_u_3312_a_fail_to_start_priority : INT;
	//Alarm delay setpoint(seconds)
	{attribute 'OPC.UA.DA' :='1'}
	popa_0081_u_3312_a_fail_to_start_delay_setpoint : INT;
	//Alarm active for HMI
	{attribute 'OPC.UA.DA' :='1'}
	popa_0081_u_3312_a_fail_to_start_active : BOOL;
	//Alarm enable
	{attribute 'OPC.UA.DA' :='1'}
	popa_0081_u_3312_a_fail_to_start_enable: BOOL;
	
	//Alarm Priority setpoint
	{attribute 'OPC.UA.DA' :='1'}
	popa_0081_u_3312_a_fail_to_stop_priority : INT;
	//Alarm delay setpoint(seconds)
	{attribute 'OPC.UA.DA' :='1'}
	popa_0081_u_3312_a_fail_to_stop_delay_setpoint : INT;
	//Alarm active for HMI
	{attribute 'OPC.UA.DA' :='1'}
	popa_0081_u_3312_a_fail_to_stop_active : BOOL;
	//Alarm enable
	{attribute 'OPC.UA.DA' :='1'}
	popa_0081_u_3312_a_fail_to_stop_enable: BOOL;
	
	//------------------------------------------------------------------------------------------------------------------
	//Alarm Priority setpoint
	{attribute 'OPC.UA.DA' :='1'}
	popa_0081_u_3160_a_fail_to_start_priority : INT;
	//Alarm delay setpoint(seconds)
	{attribute 'OPC.UA.DA' :='1'}
	popa_0081_u_3160_a_fail_to_start_delay_setpoint : INT;
	//Alarm active for HMI
	{attribute 'OPC.UA.DA' :='1'}
	popa_0081_u_3160_a_fail_to_start_active : BOOL;
	//Alarm enable
	{attribute 'OPC.UA.DA' :='1'}
	popa_0081_u_3160_a_fail_to_start_enable: BOOL;
	
	//Alarm Priority setpoint
	{attribute 'OPC.UA.DA' :='1'}
	popa_0081_u_3160_a_fail_to_stop_priority : INT;
	//Alarm delay setpoint(seconds)
	{attribute 'OPC.UA.DA' :='1'}
	popa_0081_u_3160_a_fail_to_stop_delay_setpoint : INT;
	//Alarm active for HMI
	{attribute 'OPC.UA.DA' :='1'}
	popa_0081_u_3160_a_fail_to_stop_active : BOOL;
	//Alarm enable
	{attribute 'OPC.UA.DA' :='1'}
	popa_0081_u_3160_a_fail_to_stop_enable: BOOL;
	
	//------------------------------------------------------------------------------------------------------------------
	//Alarm Priority setpoint
	{attribute 'OPC.UA.DA' :='1'}
	popa_0081_u_3260_a_fail_to_start_priority : INT;
	//Alarm delay setpoint(seconds)
	{attribute 'OPC.UA.DA' :='1'}
	popa_0081_u_3260_a_fail_to_start_delay_setpoint : INT;
	//Alarm active for HMI
	{attribute 'OPC.UA.DA' :='1'}
	popa_0081_u_3260_a_fail_to_start_active : BOOL;
	//Alarm enable
	{attribute 'OPC.UA.DA' :='1'}
	popa_0081_u_3260_a_fail_to_start_enable: BOOL;
	
	//Alarm Priority setpoint
	{attribute 'OPC.UA.DA' :='1'}
	popa_0081_u_3260_a_fail_to_stop_priority : INT;
	//Alarm delay setpoint(seconds)
	{attribute 'OPC.UA.DA' :='1'}
	popa_0081_u_3260_a_fail_to_stop_delay_setpoint : INT;
	//Alarm active for HMI
	{attribute 'OPC.UA.DA' :='1'}
	popa_0081_u_3260_a_fail_to_stop_active : BOOL;
	//Alarm enable
	{attribute 'OPC.UA.DA' :='1'}
	popa_0081_u_3260_a_fail_to_stop_enable: BOOL;
	
	//------------------------------------------------------------------------------------------------------------------
	//Alarm Priority setpoint
	{attribute 'OPC.UA.DA' :='1'}
	popa_0081_u_3360_a_fail_to_start_priority : INT;
	//Alarm delay setpoint(seconds)
	{attribute 'OPC.UA.DA' :='1'}
	popa_0081_u_3360_a_fail_to_start_delay_setpoint : INT;
	//Alarm active for HMI
	{attribute 'OPC.UA.DA' :='1'}
	popa_0081_u_3360_a_fail_to_start_active : BOOL;
	//Alarm enable
	{attribute 'OPC.UA.DA' :='1'}
	popa_0081_u_3360_a_fail_to_start_enable: BOOL;
	
	//Alarm Priority setpoint
	{attribute 'OPC.UA.DA' :='1'}
	popa_0081_u_3360_a_fail_to_stop_priority : INT;
	//Alarm delay setpoint(seconds)
	{attribute 'OPC.UA.DA' :='1'}
	popa_0081_u_3360_a_fail_to_stop_delay_setpoint : INT;
	//Alarm active for HMI
	{attribute 'OPC.UA.DA' :='1'}
	popa_0081_u_3360_a_fail_to_stop_active : BOOL;
	//Alarm enable
	{attribute 'OPC.UA.DA' :='1'}
	popa_0081_u_3360_a_fail_to_stop_enable: BOOL;
	
	//------------------------------------------------------------------------------------------------------------------
	//Alarm Priority setpoint
	{attribute 'OPC.UA.DA' :='1'}
	popa_0081_u_3370_a_fail_to_start_priority : INT;
	//Alarm delay setpoint(seconds)
	{attribute 'OPC.UA.DA' :='1'}
	popa_0081_u_3370_a_fail_to_start_delay_setpoint : INT;
	//Alarm active for HMI
	{attribute 'OPC.UA.DA' :='1'}
	popa_0081_u_3370_a_fail_to_start_active : BOOL;
	//Alarm enable
	{attribute 'OPC.UA.DA' :='1'}
	popa_0081_u_3370_a_fail_to_start_enable: BOOL;
	
	//Alarm Priority setpoint
	{attribute 'OPC.UA.DA' :='1'}
	popa_0081_u_3370_a_fail_to_stop_priority : INT;
	//Alarm delay setpoint(seconds)
	{attribute 'OPC.UA.DA' :='1'}
	popa_0081_u_3370_a_fail_to_stop_delay_setpoint : INT;
	//Alarm active for HMI
	{attribute 'OPC.UA.DA' :='1'}
	popa_0081_u_3370_a_fail_to_stop_active : BOOL;
	//Alarm enable
	{attribute 'OPC.UA.DA' :='1'}
	popa_0081_u_3370_a_fail_to_stop_enable: BOOL;
	
	//------------------------------------------------------------------------------------------------------------------
	//Alarm Priority setpoint
	{attribute 'OPC.UA.DA' :='1'}
	popa_0091_u_3405_a_fail_to_start_priority : INT;
	//Alarm delay setpoint(seconds)
	{attribute 'OPC.UA.DA' :='1'}
	popa_0091_u_3405_a_fail_to_start_delay_setpoint : INT;
	//Alarm active for HMI
	{attribute 'OPC.UA.DA' :='1'}
	popa_0091_u_3405_a_fail_to_start_active : BOOL;
	//Alarm enable
	{attribute 'OPC.UA.DA' :='1'}
	popa_0091_u_3405_a_fail_to_start_enable: BOOL;
	
	//Alarm Priority setpoint
	{attribute 'OPC.UA.DA' :='1'}
	popa_0091_u_3405_a_fail_to_stop_priority : INT;
	//Alarm delay setpoint(seconds)
	{attribute 'OPC.UA.DA' :='1'}
	popa_0091_u_3405_a_fail_to_stop_delay_setpoint : INT;
	//Alarm active for HMI
	{attribute 'OPC.UA.DA' :='1'}
	popa_0091_u_3405_a_fail_to_stop_active : BOOL;
	//Alarm enable
	{attribute 'OPC.UA.DA' :='1'}
	popa_0091_u_3405_a_fail_to_stop_enable: BOOL;

	
	//---------------------------------------------------------------------------------------------------------
	//Raw Min value for analog input
	{attribute 'OPC.UA.DA' :='1'}
	popa_0081_u_3112_a_speed_command_raw_min : REAL :=0;
	//Raw max value for analog input
	{attribute 'OPC.UA.DA' :='1'}
	popa_0081_u_3112_a_speed_command_raw_max : REAL :=32767;
	//EU Min value for analog input
	{attribute 'OPC.UA.DA' :='1'}
	popa_0081_u_3112_a_speed_command_eu_min : REAL;
	//EU Max value for analog input
	{attribute 'OPC.UA.DA' :='1'}
	popa_0081_u_3112_a_speed_command_eu_max : REAL;
	//Filter factor value for analog input
	{attribute 'OPC.UA.DA' :='1'}
	popa_0081_u_3112_a_speed_command_filter_factor : REAL;
	//Scaled value for analog input
	{attribute 'OPC.UA.DA' :='1'}
	popa_0081_u_3112_a_speed_command_scaled_value : REAL;
	
	//Raw Min value for analog input
	{attribute 'OPC.UA.DA' :='1'}
	popa_0081_u_3112_a_speed_feedback_raw_min : REAL :=0;
	//Raw max value for analog input
	{attribute 'OPC.UA.DA' :='1'}
	popa_0081_u_3112_a_speed_feedback_raw_max : REAL :=32767;
	//EU Min value for analog input
	{attribute 'OPC.UA.DA' :='1'}
	popa_0081_u_3112_a_speed_feedback_eu_min : REAL;
	//EU Max value for analog input
	{attribute 'OPC.UA.DA' :='1'}
	popa_0081_u_3112_a_speed_feedback_eu_max : REAL;
	//Filter factor value for analog input
	{attribute 'OPC.UA.DA' :='1'}
	popa_0081_u_3112_a_speed_feedback_filter_factor : REAL;
	//Scaled value for analog input
	{attribute 'OPC.UA.DA' :='1'}
	popa_0081_u_3112_a_speed_feedback_scaled_value : REAL;
	
	
	//---------------------------------------------------------------------------------------------------------
	//Raw Min value for analog input
	{attribute 'OPC.UA.DA' :='1'}
	popa_0081_u_3212_a_speed_command_raw_min : REAL :=0;
	//Raw max value for analog input
	{attribute 'OPC.UA.DA' :='1'}
	popa_0081_u_3212_a_speed_command_raw_max : REAL :=32767;
	//EU Min value for analog input
	{attribute 'OPC.UA.DA' :='1'}
	popa_0081_u_3212_a_speed_command_eu_min : REAL;
	//EU Max value for analog input
	{attribute 'OPC.UA.DA' :='1'}
	popa_0081_u_3212_a_speed_command_eu_max : REAL;
	//Filter factor value for analog input
	{attribute 'OPC.UA.DA' :='1'}
	popa_0081_u_3212_a_speed_command_filter_factor : REAL;
	//Scaled value for analog input
	{attribute 'OPC.UA.DA' :='1'}
	popa_0081_u_3212_a_speed_command_scaled_value : REAL;
	
	//Raw Min value for analog input
	{attribute 'OPC.UA.DA' :='1'}
	popa_0081_u_3212_a_speed_feedback_raw_min : REAL :=0;
	//Raw max value for analog input
	{attribute 'OPC.UA.DA' :='1'}
	popa_0081_u_3212_a_speed_feedback_raw_max : REAL :=32767;
	//EU Min value for analog input
	{attribute 'OPC.UA.DA' :='1'}
	popa_0081_u_3212_a_speed_feedback_eu_min : REAL;
	//EU Max value for analog input
	{attribute 'OPC.UA.DA' :='1'}
	popa_0081_u_3212_a_speed_feedback_eu_max : REAL;
	//Filter factor value for analog input
	{attribute 'OPC.UA.DA' :='1'}
	popa_0081_u_3212_a_speed_feedback_filter_factor : REAL;
	//Scaled value for analog input
	{attribute 'OPC.UA.DA' :='1'}
	popa_0081_u_3212_a_speed_feedback_scaled_value : REAL;
	
	
	//---------------------------------------------------------------------------------------------------------
	//Raw Min value for analog input
	{attribute 'OPC.UA.DA' :='1'}
	popa_0081_u_3312_a_speed_command_raw_min : REAL :=0;
	//Raw max value for analog input
	{attribute 'OPC.UA.DA' :='1'}
	popa_0081_u_3312_a_speed_command_raw_max : REAL :=32767;
	//EU Min value for analog input
	{attribute 'OPC.UA.DA' :='1'}
	popa_0081_u_3312_a_speed_command_eu_min : REAL;
	//EU Max value for analog input
	{attribute 'OPC.UA.DA' :='1'}
	popa_0081_u_3312_a_speed_command_eu_max : REAL;
	//Filter factor value for analog input
	{attribute 'OPC.UA.DA' :='1'}
	popa_0081_u_3312_a_speed_command_filter_factor : REAL;
	//Scaled value for analog input
	{attribute 'OPC.UA.DA' :='1'}
	popa_0081_u_3312_a_speed_command_scaled_value : REAL;
	
	//Raw Min value for analog input
	{attribute 'OPC.UA.DA' :='1'}
	popa_0081_u_3312_a_speed_feedback_raw_min : REAL :=0;
	//Raw max value for analog input
	{attribute 'OPC.UA.DA' :='1'}
	popa_0081_u_3312_a_speed_feedback_raw_max : REAL :=32767;
	//EU Min value for analog input
	{attribute 'OPC.UA.DA' :='1'}
	popa_0081_u_3312_a_speed_feedback_eu_min : REAL;
	//EU Max value for analog input
	{attribute 'OPC.UA.DA' :='1'}
	popa_0081_u_3312_a_speed_feedback_eu_max : REAL;
	//Filter factor value for analog input
	{attribute 'OPC.UA.DA' :='1'}
	popa_0081_u_3312_a_speed_feedback_filter_factor : REAL;
	//Scaled value for analog input
	{attribute 'OPC.UA.DA' :='1'}
	popa_0081_u_3312_a_speed_feedback_scaled_value : REAL;
	
	
	//---------------------------------------------------------------------------------------------------------
	//Raw Min value for analog input
	{attribute 'OPC.UA.DA' :='1'}
	popa_0081_u_3160_a_speed_command_raw_min : REAL :=0;
	//Raw max value for analog input
	{attribute 'OPC.UA.DA' :='1'}
	popa_0081_u_3160_a_speed_command_raw_max : REAL :=32767;
	//EU Min value for analog input
	{attribute 'OPC.UA.DA' :='1'}
	popa_0081_u_3160_a_speed_command_eu_min : REAL;
	//EU Max value for analog input
	{attribute 'OPC.UA.DA' :='1'}
	popa_0081_u_3160_a_speed_command_eu_max : REAL;
	//Filter factor value for analog input
	{attribute 'OPC.UA.DA' :='1'}
	popa_0081_u_3160_a_speed_command_filter_factor : REAL;
	//Scaled value for analog input
	{attribute 'OPC.UA.DA' :='1'}
	popa_0081_u_3160_a_speed_command_scaled_value : REAL;
	
	//Raw Min value for analog input
	{attribute 'OPC.UA.DA' :='1'}
	popa_0081_u_3160_a_speed_feedback_raw_min : REAL :=0;
	//Raw max value for analog input
	{attribute 'OPC.UA.DA' :='1'}
	popa_0081_u_3160_a_speed_feedback_raw_max : REAL :=32767;
	//EU Min value for analog input
	{attribute 'OPC.UA.DA' :='1'}
	popa_0081_u_3160_a_speed_feedback_eu_min : REAL;
	//EU Max value for analog input
	{attribute 'OPC.UA.DA' :='1'}
	popa_0081_u_3160_a_speed_feedback_eu_max : REAL;
	//Filter factor value for analog input
	{attribute 'OPC.UA.DA' :='1'}
	popa_0081_u_3160_a_speed_feedback_filter_factor : REAL;
	//Scaled value for analog input
	{attribute 'OPC.UA.DA' :='1'}
	popa_0081_u_3160_a_speed_feedback_scaled_value : REAL;
	
	
	//---------------------------------------------------------------------------------------------------------
	//Raw Min value for analog input
	{attribute 'OPC.UA.DA' :='1'}
	popa_0081_u_3260_a_speed_command_raw_min : REAL :=0;
	//Raw max value for analog input
	{attribute 'OPC.UA.DA' :='1'}
	popa_0081_u_3260_a_speed_command_raw_max : REAL :=32767;
	//EU Min value for analog input
	{attribute 'OPC.UA.DA' :='1'}
	popa_0081_u_3260_a_speed_command_eu_min : REAL;
	//EU Max value for analog input
	{attribute 'OPC.UA.DA' :='1'}
	popa_0081_u_3260_a_speed_command_eu_max : REAL;
	//Filter factor value for analog input
	{attribute 'OPC.UA.DA' :='1'}
	popa_0081_u_3260_a_speed_command_filter_factor : REAL;
	//Scaled value for analog input
	{attribute 'OPC.UA.DA' :='1'}
	popa_0081_u_3260_a_speed_command_scaled_value : REAL;
	
	//Raw Min value for analog input
	{attribute 'OPC.UA.DA' :='1'}
	popa_0081_u_3260_a_speed_feedback_raw_min : REAL :=0;
	//Raw max value for analog input
	{attribute 'OPC.UA.DA' :='1'}
	popa_0081_u_3260_a_speed_feedback_raw_max : REAL :=32767;
	//EU Min value for analog input
	{attribute 'OPC.UA.DA' :='1'}
	popa_0081_u_3260_a_speed_feedback_eu_min : REAL;
	//EU Max value for analog input
	{attribute 'OPC.UA.DA' :='1'}
	popa_0081_u_3260_a_speed_feedback_eu_max : REAL;
	//Filter factor value for analog input
	{attribute 'OPC.UA.DA' :='1'}
	popa_0081_u_3260_a_speed_feedback_filter_factor : REAL;
	//Scaled value for analog input
	{attribute 'OPC.UA.DA' :='1'}
	popa_0081_u_3260_a_speed_feedback_scaled_value : REAL;
	
	
	//---------------------------------------------------------------------------------------------------------
	//Raw Min value for analog input
	{attribute 'OPC.UA.DA' :='1'}
	popa_0081_u_3360_a_speed_command_raw_min : REAL :=0;
	//Raw max value for analog input
	{attribute 'OPC.UA.DA' :='1'}
	popa_0081_u_3360_a_speed_command_raw_max : REAL :=32767;
	//EU Min value for analog input
	{attribute 'OPC.UA.DA' :='1'}
	popa_0081_u_3360_a_speed_command_eu_min : REAL;
	//EU Max value for analog input
	{attribute 'OPC.UA.DA' :='1'}
	popa_0081_u_3360_a_speed_command_eu_max : REAL;
	//Filter factor value for analog input
	{attribute 'OPC.UA.DA' :='1'}
	popa_0081_u_3360_a_speed_command_filter_factor : REAL;
	//Scaled value for analog input
	{attribute 'OPC.UA.DA' :='1'}
	popa_0081_u_3360_a_speed_command_scaled_value : REAL;
	
	//Raw Min value for analog input
	{attribute 'OPC.UA.DA' :='1'}
	popa_0081_u_3360_a_speed_feedback_raw_min : REAL :=0;
	//Raw max value for analog input
	{attribute 'OPC.UA.DA' :='1'}
	popa_0081_u_3360_a_speed_feedback_raw_max : REAL :=32767;
	//EU Min value for analog input
	{attribute 'OPC.UA.DA' :='1'}
	popa_0081_u_3360_a_speed_feedback_eu_min : REAL;
	//EU Max value for analog input
	{attribute 'OPC.UA.DA' :='1'}
	popa_0081_u_3360_a_speed_feedback_eu_max : REAL;
	//Filter factor value for analog input
	{attribute 'OPC.UA.DA' :='1'}
	popa_0081_u_3360_a_speed_feedback_filter_factor : REAL;
	//Scaled value for analog input
	{attribute 'OPC.UA.DA' :='1'}
	popa_0081_u_3360_a_speed_feedback_scaled_value : REAL;
	
	
	//---------------------------------------------------------------------------------------------------------
	//Raw Min value for analog input
	{attribute 'OPC.UA.DA' :='1'}
	popa_0081_u_3370_a_speed_command_raw_min : REAL :=0;
	//Raw max value for analog input
	{attribute 'OPC.UA.DA' :='1'}
	popa_0081_u_3370_a_speed_command_raw_max : REAL :=32767;
	//EU Min value for analog input
	{attribute 'OPC.UA.DA' :='1'}
	popa_0081_u_3370_a_speed_command_eu_min : REAL;
	//EU Max value for analog input
	{attribute 'OPC.UA.DA' :='1'}
	popa_0081_u_3370_a_speed_command_eu_max : REAL;
	//Filter factor value for analog input
	{attribute 'OPC.UA.DA' :='1'}
	popa_0081_u_3370_a_speed_command_filter_factor : REAL;
	//Scaled value for analog input
	{attribute 'OPC.UA.DA' :='1'}
	popa_0081_u_3370_a_speed_command_scaled_value : REAL;
	
	//Raw Min value for analog input
	{attribute 'OPC.UA.DA' :='1'}
	popa_0081_u_3370_a_speed_feedback_raw_min : REAL :=0;
	//Raw max value for analog input
	{attribute 'OPC.UA.DA' :='1'}
	popa_0081_u_3370_a_speed_feedback_raw_max : REAL :=32767;
	//EU Min value for analog input
	{attribute 'OPC.UA.DA' :='1'}
	popa_0081_u_3370_a_speed_feedback_eu_min : REAL;
	//EU Max value for analog input
	{attribute 'OPC.UA.DA' :='1'}
	popa_0081_u_3370_a_speed_feedback_eu_max : REAL;
	//Filter factor value for analog input
	{attribute 'OPC.UA.DA' :='1'}
	popa_0081_u_3370_a_speed_feedback_filter_factor : REAL;
	//Scaled value for analog input
	{attribute 'OPC.UA.DA' :='1'}
	popa_0081_u_3370_a_speed_feedback_scaled_value : REAL;
	
	
	//---------------------------------------------------------------------------------------------------------
	//Raw Min value for analog input
	{attribute 'OPC.UA.DA' :='1'}
	popa_0091_u_3405_a_speed_command_raw_min : REAL :=0;
	//Raw max value for analog input
	{attribute 'OPC.UA.DA' :='1'}
	popa_0091_u_3405_a_speed_command_raw_max : REAL :=32767;
	//EU Min value for analog input
	{attribute 'OPC.UA.DA' :='1'}
	popa_0091_u_3405_a_speed_command_eu_min : REAL;
	//EU Max value for analog input
	{attribute 'OPC.UA.DA' :='1'}
	popa_0091_u_3405_a_speed_command_eu_max : REAL;
	//Filter factor value for analog input
	{attribute 'OPC.UA.DA' :='1'}
	popa_0091_u_3405_a_speed_command_filter_factor : REAL;
	//Scaled value for analog input
	{attribute 'OPC.UA.DA' :='1'}
	popa_0091_u_3405_a_speed_command_scaled_value : REAL;
	
	//Raw Min value for analog input
	{attribute 'OPC.UA.DA' :='1'}
	popa_0091_u_3405_a_speed_feedback_raw_min : REAL :=0;
	//Raw max value for analog input
	{attribute 'OPC.UA.DA' :='1'}
	popa_0091_u_3405_a_speed_feedback_raw_max : REAL :=32767;
	//EU Min value for analog input
	{attribute 'OPC.UA.DA' :='1'}
	popa_0091_u_3405_a_speed_feedback_eu_min : REAL;
	//EU Max value for analog input
	{attribute 'OPC.UA.DA' :='1'}
	popa_0091_u_3405_a_speed_feedback_eu_max : REAL;
	//Filter factor value for analog input
	{attribute 'OPC.UA.DA' :='1'}
	popa_0091_u_3405_a_speed_feedback_filter_factor : REAL;
	//Scaled value for analog input
	{attribute 'OPC.UA.DA' :='1'}
	popa_0091_u_3405_a_speed_feedback_scaled_value : REAL;
	
//---Valves----------------------------------------------------------------------------------------------------------------------------------------

	//Raw Min value for analog input
	{attribute 'OPC.UA.DA' :='1'}
	popa_0081_av_3148_a_position_feedback_raw_min : REAL :=0;
	//Raw max value for analog input
	{attribute 'OPC.UA.DA' :='1'}
	popa_0081_av_3148_a_position_feedback_raw_max : REAL :=32767;
	//EU Min value for analog input
	{attribute 'OPC.UA.DA' :='1'}
	popa_0081_av_3148_a_position_feedback_eu_min : REAL;
	//EU Max value for analog input
	{attribute 'OPC.UA.DA' :='1'}
	popa_0081_av_3148_a_position_feedback_eu_max : REAL;
	//Filter factor value for analog input
	{attribute 'OPC.UA.DA' :='1'}
	popa_0081_av_3148_a_position_feedback_filter_factor : REAL;
	//Scaled value for analog input
	{attribute 'OPC.UA.DA' :='1'}
	popa_0081_av_3148_a_position_feedback_scaled_value : REAL;
	
	//Raw Min value for analog input
	{attribute 'OPC.UA.DA' :='1'}
	popa_0081_av_3148_a_position_command_raw_min : REAL :=0;
	//Raw max value for analog input
	{attribute 'OPC.UA.DA' :='1'}
	popa_0081_av_3148_a_position_command_raw_max : REAL :=32767;
	//EU Min value for analog input
	{attribute 'OPC.UA.DA' :='1'}
	popa_0081_av_3148_a_position_command_eu_min : REAL;
	//EU Max value for analog input
	{attribute 'OPC.UA.DA' :='1'}
	popa_0081_av_3148_a_position_command_eu_max : REAL;
	//Filter factor value for analog input
	{attribute 'OPC.UA.DA' :='1'}
	popa_0081_av_3148_a_position_command_filter_factor : REAL;
	//Scaled value for analog input
	{attribute 'OPC.UA.DA' :='1'}
	popa_0081_av_3148_a_position_command_scaled_value : REAL;
//-----------------------------------------------------------------------------------------------------------	
	//Raw Min value for analog input
	{attribute 'OPC.UA.DA' :='1'}
	popa_0081_av_3248_a_position_feedback_raw_min : REAL :=0;
	//Raw max value for analog input
	{attribute 'OPC.UA.DA' :='1'}
	popa_0081_av_3248_a_position_feedback_raw_max : REAL :=32767;
	//EU Min value for analog input
	{attribute 'OPC.UA.DA' :='1'}
	popa_0081_av_3248_a_position_feedback_eu_min : REAL;
	//EU Max value for analog input
	{attribute 'OPC.UA.DA' :='1'}
	popa_0081_av_3248_a_position_feedback_eu_max : REAL;
	//Filter factor value for analog input
	{attribute 'OPC.UA.DA' :='1'}
	popa_0081_av_3248_a_position_feedback_filter_factor : REAL;
	//Scaled value for analog input
	{attribute 'OPC.UA.DA' :='1'}
	popa_0081_av_3248_a_position_feedback_scaled_value : REAL;
	
	//Raw Min value for analog input
	{attribute 'OPC.UA.DA' :='1'}
	popa_0081_av_3248_a_position_command_raw_min : REAL :=0;
	//Raw max value for analog input
	{attribute 'OPC.UA.DA' :='1'}
	popa_0081_av_3248_a_position_command_raw_max : REAL :=32767;
	//EU Min value for analog input
	{attribute 'OPC.UA.DA' :='1'}
	popa_0081_av_3248_a_position_command_eu_min : REAL;
	//EU Max value for analog input
	{attribute 'OPC.UA.DA' :='1'}
	popa_0081_av_3248_a_position_command_eu_max : REAL;
	//Filter factor value for analog input
	{attribute 'OPC.UA.DA' :='1'}
	popa_0081_av_3248_a_position_command_filter_factor : REAL;
	//Scaled value for analog input
	{attribute 'OPC.UA.DA' :='1'}
	popa_0081_av_3248_a_position_command_scaled_value : REAL;
//-----------------------------------------------------------------------------------------------------------	

	//Raw Min value for analog input
	{attribute 'OPC.UA.DA' :='1'}
	popa_0081_av_3348_a_position_feedback_raw_min : REAL :=0;
	//Raw max value for analog input
	{attribute 'OPC.UA.DA' :='1'}
	popa_0081_av_3348_a_position_feedback_raw_max : REAL :=32767;
	//EU Min value for analog input
	{attribute 'OPC.UA.DA' :='1'}
	popa_0081_av_3348_a_position_feedback_eu_min : REAL;
	//EU Max value for analog input
	{attribute 'OPC.UA.DA' :='1'}
	popa_0081_av_3348_a_position_feedback_eu_max : REAL;
	//Filter factor value for analog input
	{attribute 'OPC.UA.DA' :='1'}
	popa_0081_av_3348_a_position_feedback_filter_factor : REAL;
	//Scaled value for analog input
	{attribute 'OPC.UA.DA' :='1'}
	popa_0081_av_3348_a_position_feedback_scaled_value : REAL;
	
	//Raw Min value for analog input
	{attribute 'OPC.UA.DA' :='1'}
	popa_0081_av_3348_a_position_command_raw_min : REAL :=0;
	//Raw max value for analog input
	{attribute 'OPC.UA.DA' :='1'}
	popa_0081_av_3348_a_position_command_raw_max : REAL :=32767;
	//EU Min value for analog input
	{attribute 'OPC.UA.DA' :='1'}
	popa_0081_av_3348_a_position_command_eu_min : REAL;
	//EU Max value for analog input
	{attribute 'OPC.UA.DA' :='1'}
	popa_0081_av_3348_a_position_command_eu_max : REAL;
	//Filter factor value for analog input
	{attribute 'OPC.UA.DA' :='1'}
	popa_0081_av_3348_a_position_command_filter_factor : REAL;
	//Scaled value for analog input
	{attribute 'OPC.UA.DA' :='1'}
	popa_0081_av_3348_a_position_command_scaled_value : REAL;
//-----------------------------------------------------------------------------------------------------------		


	//Example motor starter runtime maintenance reset
	{attribute 'OPC.UA.DA' :='1'}
	popa_0081_u_3160_a_runtime_maint_reset : BOOL;
	//Example motor starter run request
	{attribute 'OPC.UA.DA' :='1'}
	popa_0081_u_3160_a_run_request : BOOL;
	//Example motor starter runtime today
	{attribute 'OPC.UA.DA' :='1'}
	popa_0081_u_3160_a_runtime_today : REAL;
	//Example motor starter runtime total
	{attribute 'OPC.UA.DA' :='1'}
	popa_0081_u_3160_a_runtime_total : REAL;
	//Example motor starter runtime maint
	{attribute 'OPC.UA.DA' :='1'}
	popa_0081_u_3160_a_runtime_maint : REAL;
	//Example motor starter status, 0=Off, 1=Run, 2=Fault
	{attribute 'OPC.UA.DA' :='1'}
	popa_0081_u_3160_a_status : REAL;
	
	//--------------------------------------------------------------------------------------------------------------
	//Example motor vfd runtime maintenance reset
	{attribute 'OPC.UA.DA' :='1'}
	popa_0081_u_3112_a_runtime_maint_reset : BOOL;
	//Example motor vfd run request
	{attribute 'OPC.UA.DA' :='1'}
	popa_0081_u_3112_a_run_request : BOOL;
	//Example motor vfd speed request
	{attribute 'OPC.UA.DA' :='1'}
	popa_0081_u_3112_a_speed_request : REAL;
	//Example motor vfd speed feedback
	{attribute 'OPC.UA.DA' :='1'}
	popa_0081_u_3112_a_speed_feedback : REAL;
	//Example motor vfd runtime today
	{attribute 'OPC.UA.DA' :='1'}
	popa_0081_u_3112_a_runtime_today : REAL;
	//Example motor vfd runtime total
	{attribute 'OPC.UA.DA' :='1'}
	popa_0081_u_3112_a_runtime_total : REAL;
	//Example motor vfd runtime maint
	{attribute 'OPC.UA.DA' :='1'}
	popa_0081_u_3112_a_runtime_maint : REAL;
	//Example motor vfd status, 0=Off, 1=Run, 2=Fault
	{attribute 'OPC.UA.DA' :='1'}
	popa_0081_u_3112_a_status : REAL;
	
	//--------------------------------------------------------------------------------------------------------------
	//Example motor vfd runtime maintenance reset
	{attribute 'OPC.UA.DA' :='1'}
	popa_0081_u_3212_a_runtime_maint_reset : BOOL;
	//Example motor vfd run request
	{attribute 'OPC.UA.DA' :='1'}
	popa_0081_u_3212_a_run_request : BOOL;
	//Example motor vfd speed request
	{attribute 'OPC.UA.DA' :='1'}
	popa_0081_u_3212_a_speed_request : REAL;
	//Example motor vfd speed feedback
	{attribute 'OPC.UA.DA' :='1'}
	popa_0081_u_3212_a_speed_feedback : REAL;
	//Example motor vfd runtime today
	{attribute 'OPC.UA.DA' :='1'}
	popa_0081_u_3212_a_runtime_today : REAL;
	//Example motor vfd runtime total
	{attribute 'OPC.UA.DA' :='1'}
	popa_0081_u_3212_a_runtime_total : REAL;
	//Example motor vfd runtime maint
	{attribute 'OPC.UA.DA' :='1'}
	popa_0081_u_3212_a_runtime_maint : REAL;
	//Example motor vfd status, 0=Off, 1=Run, 2=Fault
	{attribute 'OPC.UA.DA' :='1'}
	popa_0081_u_3212_a_status : REAL;
	
	//--------------------------------------------------------------------------------------------------------------
	//Example motor vfd runtime maintenance reset
	{attribute 'OPC.UA.DA' :='1'}
	popa_0081_u_3312_a_runtime_maint_reset : BOOL;
	//Example motor vfd run request
	{attribute 'OPC.UA.DA' :='1'}
	popa_0081_u_3312_a_run_request : BOOL;
	//Example motor vfd speed request
	{attribute 'OPC.UA.DA' :='1'}
	popa_0081_u_3312_a_speed_request : REAL;
	//Example motor vfd speed feedback
	{attribute 'OPC.UA.DA' :='1'}
	popa_0081_u_3312_a_speed_feedback : REAL;
	//Example motor vfd runtime today
	{attribute 'OPC.UA.DA' :='1'}
	popa_0081_u_3312_a_runtime_today : REAL;
	//Example motor vfd runtime total
	{attribute 'OPC.UA.DA' :='1'}
	popa_0081_u_3312_a_runtime_total : REAL;
	//Example motor vfd runtime maint
	{attribute 'OPC.UA.DA' :='1'}
	popa_0081_u_3312_a_runtime_maint : REAL;
	//Example motor vfd status, 0=Off, 1=Run, 2=Fault
	{attribute 'OPC.UA.DA' :='1'}
	popa_0081_u_3312_a_status : REAL;
	
	//--------------------------------------------------------------------------------------------------------------
	
	//Example motor vfd speed request
	{attribute 'OPC.UA.DA' :='1'}
	popa_0081_u_3160_a_speed_request : REAL;
	//Example motor vfd speed feedback
	{attribute 'OPC.UA.DA' :='1'}
	popa_0081_u_3160_a_speed_feedback : REAL;

	
	
	//--------------------------------------------------------------------------------------------------------------
	//Example motor vfd runtime maintenance reset
	{attribute 'OPC.UA.DA' :='1'}
	popa_0081_u_3260_a_runtime_maint_reset : BOOL;
	//Example motor vfd run request
	{attribute 'OPC.UA.DA' :='1'}
	popa_0081_u_3260_a_run_request : BOOL;
	//Example motor vfd speed request
	{attribute 'OPC.UA.DA' :='1'}
	popa_0081_u_3260_a_speed_request : REAL;
	//Example motor vfd speed feedback
	{attribute 'OPC.UA.DA' :='1'}
	popa_0081_u_3260_a_speed_feedback : REAL;
	//Example motor vfd runtime today
	{attribute 'OPC.UA.DA' :='1'}
	popa_0081_u_3260_a_runtime_today : REAL;
	//Example motor vfd runtime total
	{attribute 'OPC.UA.DA' :='1'}
	popa_0081_u_3260_a_runtime_total : REAL;
	//Example motor vfd runtime maint
	{attribute 'OPC.UA.DA' :='1'}
	popa_0081_u_3260_a_runtime_maint : REAL;
	//Example motor vfd status, 0=Off, 1=Run, 2=Fault
	{attribute 'OPC.UA.DA' :='1'}
	popa_0081_u_3260_a_status : REAL;
	
	//--------------------------------------------------------------------------------------------------------------
	//Example motor vfd runtime maintenance reset
	{attribute 'OPC.UA.DA' :='1'}
	popa_0081_u_3360_a_runtime_maint_reset : BOOL;
	//Example motor vfd run request
	{attribute 'OPC.UA.DA' :='1'}
	popa_0081_u_3360_a_run_request : BOOL;
	//Example motor vfd speed request
	{attribute 'OPC.UA.DA' :='1'}
	popa_0081_u_3360_a_speed_request : REAL;
	//Example motor vfd speed feedback
	{attribute 'OPC.UA.DA' :='1'}
	popa_0081_u_3360_a_speed_feedback : REAL;
	//Example motor vfd runtime today
	{attribute 'OPC.UA.DA' :='1'}
	popa_0081_u_3360_a_runtime_today : REAL;
	//Example motor vfd runtime total
	{attribute 'OPC.UA.DA' :='1'}
	popa_0081_u_3360_a_runtime_total : REAL;
	//Example motor vfd runtime maint
	{attribute 'OPC.UA.DA' :='1'}
	popa_0081_u_3360_a_runtime_maint : REAL;
	//Example motor vfd status, 0=Off, 1=Run, 2=Fault
	{attribute 'OPC.UA.DA' :='1'}
	popa_0081_u_3360_a_status : REAL;
	
	//--------------------------------------------------------------------------------------------------------------
	//Example motor vfd runtime maintenance reset
	{attribute 'OPC.UA.DA' :='1'}
	popa_0081_u_3370_a_runtime_maint_reset : BOOL;
	//Example motor vfd run request
	{attribute 'OPC.UA.DA' :='1'}
	popa_0081_u_3370_a_run_request : BOOL;
	//Example motor vfd speed request
	{attribute 'OPC.UA.DA' :='1'}
	popa_0081_u_3370_a_speed_request : REAL;
	//Example motor vfd speed feedback
	{attribute 'OPC.UA.DA' :='1'}
	popa_0081_u_3370_a_speed_feedback : REAL;
	//Example motor vfd runtime today
	{attribute 'OPC.UA.DA' :='1'}
	popa_0081_u_3370_a_runtime_today : REAL;
	//Example motor vfd runtime total
	{attribute 'OPC.UA.DA' :='1'}
	popa_0081_u_3370_a_runtime_total : REAL;
	//Example motor vfd runtime maint
	{attribute 'OPC.UA.DA' :='1'}
	popa_0081_u_3370_a_runtime_maint : REAL;
	//Example motor vfd status, 0=Off, 1=Run, 2=Fault
	{attribute 'OPC.UA.DA' :='1'}
	popa_0081_u_3370_a_status : REAL;
	
	//--------------------------------------------------------------------------------------------------------------
	//Example motor vfd runtime maintenance reset
	{attribute 'OPC.UA.DA' :='1'}
	popa_0091_u_3405_a_runtime_maint_reset : BOOL;
	//Example motor vfd run request
	{attribute 'OPC.UA.DA' :='1'}
	popa_0091_u_3405_a_run_request : BOOL;
	//Example motor vfd speed request
	{attribute 'OPC.UA.DA' :='1'}
	popa_0091_u_3405_a_speed_request : REAL;
	//Example motor vfd speed feedback
	{attribute 'OPC.UA.DA' :='1'}
	popa_0091_u_3405_a_speed_feedback : REAL;
	//Example motor vfd runtime today
	{attribute 'OPC.UA.DA' :='1'}
	popa_0091_u_3405_a_runtime_today : REAL;
	//Example motor vfd runtime total
	{attribute 'OPC.UA.DA' :='1'}
	popa_0091_u_3405_a_runtime_total : REAL;
	//Example motor vfd runtime maint
	{attribute 'OPC.UA.DA' :='1'}
	popa_0091_u_3405_a_runtime_maint : REAL;
	//Example motor vfd status, 0=Off, 1=Run, 2=Fault
	{attribute 'OPC.UA.DA' :='1'}
	popa_0091_u_3405_a_status : REAL;
	
	
	//Analog valve position request
	{attribute 'OPC.UA.DA' :='1'}
	popa_0081_av_3148_a_position_feedback : REAL;
	//Example analog valve position request
	{attribute 'OPC.UA.DA' :='1'}
	popa_0081_av_3148_a_position_request : REAL;
	//Example analog valve position fail deadband
	{attribute 'OPC.UA.DA' :='1'}
	popa_0081_av_3148_a_position_deadband_sp : REAL;
	//Example analog valve position requested when in fault state
	{attribute 'OPC.UA.DA' :='1'}
	popa_0081_av_3148_a_position_faulted : REAL;
	//Example analog valve status
	{attribute 'OPC.UA.DA' :='1'}
	popa_0081_av_3148_a_status : INT;
	//-------------------------------------------------------------------------------------------
		{attribute 'OPC.UA.DA' :='1'}
	popa_0081_av_3248_a_position_feedback : REAL;
	//Example analog valve position request
	{attribute 'OPC.UA.DA' :='1'}
	popa_0081_av_3248_a_position_request : REAL;
	//Example analog valve position fail deadband
	{attribute 'OPC.UA.DA' :='1'}
	popa_0081_av_3248_a_position_deadband_sp : REAL;
	//Example analog valve position requested when in fault state
	{attribute 'OPC.UA.DA' :='1'}
	popa_0081_av_3248_a_position_faulted : REAL;
	//Example analog valve status
	{attribute 'OPC.UA.DA' :='1'}
	popa_0081_av_3248_a_status : INT;
	//-------------------------------------------------------------------------------------------
		{attribute 'OPC.UA.DA' :='1'}
	popa_0081_av_3348_a_position_feedback : REAL;
	//Example analog valve position request
	{attribute 'OPC.UA.DA' :='1'}
	popa_0081_av_3348_a_position_request : REAL;
	//Example analog valve position fail deadband
	{attribute 'OPC.UA.DA' :='1'}
	popa_0081_av_3348_a_position_deadband_sp : REAL;
	//Example analog valve position requested when in fault state
	{attribute 'OPC.UA.DA' :='1'}
	popa_0081_av_3348_a_position_faulted : REAL;
	//Example analog valve status
	{attribute 'OPC.UA.DA' :='1'}
	popa_0081_av_3348_a_status : INT;
	
	
	
	
//---Sensors----------------------------------------------------------------------------------------------------------------------------	
	//---cpt_3144-----------------------------------------------------------------------------------------------------------------------
	//Alarm Priority setpoint
	{attribute 'OPC.UA.DA' :='1'}
	popa_0081_cpt_3144_a_low_low_priority : INT;
	//Alarm delay setpoint(seconds)
	{attribute 'OPC.UA.DA' :='1'}
	popa_0081_cpt_3144_a_low_low_delay_setpoint : INT;
	//Alarm active for HMI
	{attribute 'OPC.UA.DA' :='1'}
	popa_0081_cpt_3144_a_low_low_active : BOOL;
	//Analog Alarm Setpoint
	{attribute 'OPC.UA.DA' :='1'}
	popa_0081_cpt_3144_a_low_low_setpoint : REAL;
	//Alarm enable
	{attribute 'OPC.UA.DA' :='1'}
	popa_0081_cpt_3144_a_low_low_enable: BOOL;
	
	//Alarm Priority setpoint
	{attribute 'OPC.UA.DA' :='1'}
	popa_0081_cpt_3144_a_low_priority : INT;
	//Alarm delay setpoint(seconds)
	{attribute 'OPC.UA.DA' :='1'}
	popa_0081_cpt_3144_a_low_delay_setpoint : INT;
	//Alarm active for HMI
	{attribute 'OPC.UA.DA' :='1'}
	popa_0081_cpt_3144_a_low_active : BOOL;
	//Analog Alarm Setpoint
	{attribute 'OPC.UA.DA' :='1'}
	popa_0081_cpt_3144_a_low_setpoint : REAL;
	//Alarm enable
	{attribute 'OPC.UA.DA' :='1'}
	popa_0081_cpt_3144_a_low_enable: BOOL;
	
	//Alarm Priority setpoint
	{attribute 'OPC.UA.DA' :='1'}
	popa_0081_cpt_3144_a_high_priority : INT;
	//Alarm delay setpoint(seconds)
	{attribute 'OPC.UA.DA' :='1'}
	popa_0081_cpt_3144_a_high_delay_setpoint : INT;
	//Alarm active for HMI
	{attribute 'OPC.UA.DA' :='1'}
	popa_0081_cpt_3144_a_high_active : BOOL;
	//Analog Alarm Setpoint
	{attribute 'OPC.UA.DA' :='1'}
	popa_0081_cpt_3144_a_high_setpoint : REAL;
	//Alarm enable
	{attribute 'OPC.UA.DA' :='1'}
	popa_0081_cpt_3144_a_high_enable: BOOL;
	
	//Alarm Priority setpoint
	{attribute 'OPC.UA.DA' :='1'}
	popa_0081_cpt_3144_a_high_high_priority : INT;
	//Alarm delay setpoint(seconds)
	{attribute 'OPC.UA.DA' :='1'}
	popa_0081_cpt_3144_a_high_high_delay_setpoint : INT;
	//Alarm active for HMI
	{attribute 'OPC.UA.DA' :='1'}
	popa_0081_cpt_3144_a_high_high_active : BOOL;
	//Analog Alarm Setpoint
	{attribute 'OPC.UA.DA' :='1'}
	popa_0081_cpt_3144_a_high_high_setpoint : REAL;
	//Alarm enable
	{attribute 'OPC.UA.DA' :='1'}
	popa_0081_cpt_3144_a_high_high_enable: BOOL;
	
	
	//Raw Min value for analog input
	{attribute 'OPC.UA.DA' :='1'}
	popa_0081_cpt_3144_a_raw_min : REAL :=0;
	//Raw max value for analog input
	{attribute 'OPC.UA.DA' :='1'}
	popa_0081_cpt_3144_a_raw_max : REAL :=32767;
	//EU Min value for analog input
	{attribute 'OPC.UA.DA' :='1'}
	popa_0081_cpt_3144_a_eu_min : REAL;
	//EU Max value for analog input
	{attribute 'OPC.UA.DA' :='1'}
	popa_0081_cpt_3144_a_eu_max : REAL;
	//Filter factor value for analog input
	{attribute 'OPC.UA.DA' :='1'}
	popa_0081_cpt_3144_a_filter_factor : REAL;
	//Scaled value for analog input
	{attribute 'OPC.UA.DA' :='1'}
	popa_0081_cpt_3144_a_scaled_value : REAL;
	
	//---cct_3120-----------------------------------------------------------------------------------------------------------------------
	//Alarm Priority setpoint
	{attribute 'OPC.UA.DA' :='1'}
	popa_0081_cct_3120_a_low_low_priority : INT;
	//Alarm delay setpoint(seconds)
	{attribute 'OPC.UA.DA' :='1'}
	popa_0081_cct_3120_a_low_low_delay_setpoint : INT;
	//Alarm active for HMI
	{attribute 'OPC.UA.DA' :='1'}
	popa_0081_cct_3120_a_low_low_active : BOOL;
	//Analog Alarm Setpoint
	{attribute 'OPC.UA.DA' :='1'}
	popa_0081_cct_3120_a_low_low_setpoint : REAL;
	//Alarm enable
	{attribute 'OPC.UA.DA' :='1'}
	popa_0081_cct_3120_a_low_low_enable: BOOL;
	
	//Alarm Priority setpoint
	{attribute 'OPC.UA.DA' :='1'}
	popa_0081_cct_3120_a_low_priority : INT;
	//Alarm delay setpoint(seconds)
	{attribute 'OPC.UA.DA' :='1'}
	popa_0081_cct_3120_a_low_delay_setpoint : INT;
	//Alarm active for HMI
	{attribute 'OPC.UA.DA' :='1'}
	popa_0081_cct_3120_a_low_active : BOOL;
	//Analog Alarm Setpoint
	{attribute 'OPC.UA.DA' :='1'}
	popa_0081_cct_3120_a_low_setpoint : REAL;
	//Alarm enable
	{attribute 'OPC.UA.DA' :='1'}
	popa_0081_cct_3120_a_low_enable: BOOL;
	
	//Alarm Priority setpoint
	{attribute 'OPC.UA.DA' :='1'}
	popa_0081_cct_3120_a_high_priority : INT;
	//Alarm delay setpoint(seconds)
	{attribute 'OPC.UA.DA' :='1'}
	popa_0081_cct_3120_a_high_delay_setpoint : INT;
	//Alarm active for HMI
	{attribute 'OPC.UA.DA' :='1'}
	popa_0081_cct_3120_a_high_active : BOOL;
	//Analog Alarm Setpoint
	{attribute 'OPC.UA.DA' :='1'}
	popa_0081_cct_3120_a_high_setpoint : REAL;
	//Alarm enable
	{attribute 'OPC.UA.DA' :='1'}
	popa_0081_cct_3120_a_high_enable: BOOL;
	
	//Alarm Priority setpoint
	{attribute 'OPC.UA.DA' :='1'}
	popa_0081_cct_3120_a_high_high_priority : INT;
	//Alarm delay setpoint(seconds)
	{attribute 'OPC.UA.DA' :='1'}
	popa_0081_cct_3120_a_high_high_delay_setpoint : INT;
	//Alarm active for HMI
	{attribute 'OPC.UA.DA' :='1'}
	popa_0081_cct_3120_a_high_high_active : BOOL;
	//Analog Alarm Setpoint
	{attribute 'OPC.UA.DA' :='1'}
	popa_0081_cct_3120_a_high_high_setpoint : REAL;
	//Alarm enable
	{attribute 'OPC.UA.DA' :='1'}
	popa_0081_cct_3120_a_high_high_enable: BOOL;
	
	
	//Raw Min value for analog input
	{attribute 'OPC.UA.DA' :='1'}
	popa_0081_cct_3120_a_raw_min : REAL :=0;
	//Raw max value for analog input
	{attribute 'OPC.UA.DA' :='1'}
	popa_0081_cct_3120_a_raw_max : REAL :=32767;
	//EU Min value for analog input
	{attribute 'OPC.UA.DA' :='1'}
	popa_0081_cct_3120_a_eu_min : REAL;
	//EU Max value for analog input
	{attribute 'OPC.UA.DA' :='1'}
	popa_0081_cct_3120_a_eu_max : REAL;
	//Filter factor value for analog input
	{attribute 'OPC.UA.DA' :='1'}
	popa_0081_cct_3120_a_filter_factor : REAL;
	//Scaled value for analog input
	{attribute 'OPC.UA.DA' :='1'}
	popa_0081_cct_3120_a_scaled_value : REAL;
	
		//---cct_3220-----------------------------------------------------------------------------------------------------------------------
	//Alarm Priority setpoint
	{attribute 'OPC.UA.DA' :='1'}
	popa_0081_cct_3220_a_low_low_priority : INT;
	//Alarm delay setpoint(seconds)
	{attribute 'OPC.UA.DA' :='1'}
	popa_0081_cct_3220_a_low_low_delay_setpoint : INT;
	//Alarm active for HMI
	{attribute 'OPC.UA.DA' :='1'}
	popa_0081_cct_3220_a_low_low_active : BOOL;
	//Analog Alarm Setpoint
	{attribute 'OPC.UA.DA' :='1'}
	popa_0081_cct_3220_a_low_low_setpoint : REAL;
	//Alarm enable
	{attribute 'OPC.UA.DA' :='1'}
	popa_0081_cct_3220_a_low_low_enable: BOOL;
	
	//Alarm Priority setpoint
	{attribute 'OPC.UA.DA' :='1'}
	popa_0081_cct_3220_a_low_priority : INT;
	//Alarm delay setpoint(seconds)
	{attribute 'OPC.UA.DA' :='1'}
	popa_0081_cct_3220_a_low_delay_setpoint : INT;
	//Alarm active for HMI
	{attribute 'OPC.UA.DA' :='1'}
	popa_0081_cct_3220_a_low_active : BOOL;
	//Analog Alarm Setpoint
	{attribute 'OPC.UA.DA' :='1'}
	popa_0081_cct_3220_a_low_setpoint : REAL;
	//Alarm enable
	{attribute 'OPC.UA.DA' :='1'}
	popa_0081_cct_3220_a_low_enable: BOOL;
	
	//Alarm Priority setpoint
	{attribute 'OPC.UA.DA' :='1'}
	popa_0081_cct_3220_a_high_priority : INT;
	//Alarm delay setpoint(seconds)
	{attribute 'OPC.UA.DA' :='1'}
	popa_0081_cct_3220_a_high_delay_setpoint : INT;
	//Alarm active for HMI
	{attribute 'OPC.UA.DA' :='1'}
	popa_0081_cct_3220_a_high_active : BOOL;
	//Analog Alarm Setpoint
	{attribute 'OPC.UA.DA' :='1'}
	popa_0081_cct_3220_a_high_setpoint : REAL;
	//Alarm enable
	{attribute 'OPC.UA.DA' :='1'}
	popa_0081_cct_3220_a_high_enable: BOOL;
	
	//Alarm Priority setpoint
	{attribute 'OPC.UA.DA' :='1'}
	popa_0081_cct_3220_a_high_high_priority : INT;
	//Alarm delay setpoint(seconds)
	{attribute 'OPC.UA.DA' :='1'}
	popa_0081_cct_3220_a_high_high_delay_setpoint : INT;
	//Alarm active for HMI
	{attribute 'OPC.UA.DA' :='1'}
	popa_0081_cct_3220_a_high_high_active : BOOL;
	//Analog Alarm Setpoint
	{attribute 'OPC.UA.DA' :='1'}
	popa_0081_cct_3220_a_high_high_setpoint : REAL;
	//Alarm enable
	{attribute 'OPC.UA.DA' :='1'}
	popa_0081_cct_3220_a_high_high_enable: BOOL;
	
	
	//Raw Min value for analog input
	{attribute 'OPC.UA.DA' :='1'}
	popa_0081_cct_3220_a_raw_min : REAL :=0;
	//Raw max value for analog input
	{attribute 'OPC.UA.DA' :='1'}
	popa_0081_cct_3220_a_raw_max : REAL :=32767;
	//EU Min value for analog input
	{attribute 'OPC.UA.DA' :='1'}
	popa_0081_cct_3220_a_eu_min : REAL;
	//EU Max value for analog input
	{attribute 'OPC.UA.DA' :='1'}
	popa_0081_cct_3220_a_eu_max : REAL;
	//Filter factor value for analog input
	{attribute 'OPC.UA.DA' :='1'}
	popa_0081_cct_3220_a_filter_factor : REAL;
	//Scaled value for analog input
	{attribute 'OPC.UA.DA' :='1'}
	popa_0081_cct_3220_a_scaled_value : REAL;
	
		//---cct_3320-----------------------------------------------------------------------------------------------------------------------
	//Alarm Priority setpoint
	{attribute 'OPC.UA.DA' :='1'}
	popa_0081_cct_3320_a_low_low_priority : INT;
	//Alarm delay setpoint(seconds)
	{attribute 'OPC.UA.DA' :='1'}
	popa_0081_cct_3320_a_low_low_delay_setpoint : INT;
	//Alarm active for HMI
	{attribute 'OPC.UA.DA' :='1'}
	popa_0081_cct_3320_a_low_low_active : BOOL;
	//Analog Alarm Setpoint
	{attribute 'OPC.UA.DA' :='1'}
	popa_0081_cct_3320_a_low_low_setpoint : REAL;
	//Alarm enable
	{attribute 'OPC.UA.DA' :='1'}
	popa_0081_cct_3320_a_low_low_enable: BOOL;
	
	//Alarm Priority setpoint
	{attribute 'OPC.UA.DA' :='1'}
	popa_0081_cct_3320_a_low_priority : INT;
	//Alarm delay setpoint(seconds)
	{attribute 'OPC.UA.DA' :='1'}
	popa_0081_cct_3320_a_low_delay_setpoint : INT;
	//Alarm active for HMI
	{attribute 'OPC.UA.DA' :='1'}
	popa_0081_cct_3320_a_low_active : BOOL;
	//Analog Alarm Setpoint
	{attribute 'OPC.UA.DA' :='1'}
	popa_0081_cct_3320_a_low_setpoint : REAL;
	//Alarm enable
	{attribute 'OPC.UA.DA' :='1'}
	popa_0081_cct_3320_a_low_enable: BOOL;
	
	//Alarm Priority setpoint
	{attribute 'OPC.UA.DA' :='1'}
	popa_0081_cct_3320_a_high_priority : INT;
	//Alarm delay setpoint(seconds)
	{attribute 'OPC.UA.DA' :='1'}
	popa_0081_cct_3320_a_high_delay_setpoint : INT;
	//Alarm active for HMI
	{attribute 'OPC.UA.DA' :='1'}
	popa_0081_cct_3320_a_high_active : BOOL;
	//Analog Alarm Setpoint
	{attribute 'OPC.UA.DA' :='1'}
	popa_0081_cct_3320_a_high_setpoint : REAL;
	//Alarm enable
	{attribute 'OPC.UA.DA' :='1'}
	popa_0081_cct_3320_a_high_enable: BOOL;
	
	//Alarm Priority setpoint
	{attribute 'OPC.UA.DA' :='1'}
	popa_0081_cct_3320_a_high_high_priority : INT;
	//Alarm delay setpoint(seconds)
	{attribute 'OPC.UA.DA' :='1'}
	popa_0081_cct_3320_a_high_high_delay_setpoint : INT;
	//Alarm active for HMI
	{attribute 'OPC.UA.DA' :='1'}
	popa_0081_cct_3320_a_high_high_active : BOOL;
	//Analog Alarm Setpoint
	{attribute 'OPC.UA.DA' :='1'}
	popa_0081_cct_3320_a_high_high_setpoint : REAL;
	//Alarm enable
	{attribute 'OPC.UA.DA' :='1'}
	popa_0081_cct_3320_a_high_high_enable: BOOL;
	
	
	//Raw Min value for analog input
	{attribute 'OPC.UA.DA' :='1'}
	popa_0081_cct_3320_a_raw_min : REAL :=0;
	//Raw max value for analog input
	{attribute 'OPC.UA.DA' :='1'}
	popa_0081_cct_3320_a_raw_max : REAL :=32767;
	//EU Min value for analog input
	{attribute 'OPC.UA.DA' :='1'}
	popa_0081_cct_3320_a_eu_min : REAL;
	//EU Max value for analog input
	{attribute 'OPC.UA.DA' :='1'}
	popa_0081_cct_3320_a_eu_max : REAL;
	//Filter factor value for analog input
	{attribute 'OPC.UA.DA' :='1'}
	popa_0081_cct_3320_a_filter_factor : REAL;
	//Scaled value for analog input
	{attribute 'OPC.UA.DA' :='1'}
	popa_0081_cct_3320_a_scaled_value : REAL;
	
		//---cct_3142-----------------------------------------------------------------------------------------------------------------------
	//Alarm Priority setpoint
	{attribute 'OPC.UA.DA' :='1'}
	popa_0081_cct_3142_a_low_low_priority : INT;
	//Alarm delay setpoint(seconds)
	{attribute 'OPC.UA.DA' :='1'}
	popa_0081_cct_3142_a_low_low_delay_setpoint : INT;
	//Alarm active for HMI
	{attribute 'OPC.UA.DA' :='1'}
	popa_0081_cct_3142_a_low_low_active : BOOL;
	//Analog Alarm Setpoint
	{attribute 'OPC.UA.DA' :='1'}
	popa_0081_cct_3142_a_low_low_setpoint : REAL;
	//Alarm enable
	{attribute 'OPC.UA.DA' :='1'}
	popa_0081_cct_3142_a_low_low_enable: BOOL;
	
	//Alarm Priority setpoint
	{attribute 'OPC.UA.DA' :='1'}
	popa_0081_cct_3142_a_low_priority : INT;
	//Alarm delay setpoint(seconds)
	{attribute 'OPC.UA.DA' :='1'}
	popa_0081_cct_3142_a_low_delay_setpoint : INT;
	//Alarm active for HMI
	{attribute 'OPC.UA.DA' :='1'}
	popa_0081_cct_3142_a_low_active : BOOL;
	//Analog Alarm Setpoint
	{attribute 'OPC.UA.DA' :='1'}
	popa_0081_cct_3142_a_low_setpoint : REAL;
	//Alarm enable
	{attribute 'OPC.UA.DA' :='1'}
	popa_0081_cct_3142_a_low_enable: BOOL;
	
	//Alarm Priority setpoint
	{attribute 'OPC.UA.DA' :='1'}
	popa_0081_cct_3142_a_high_priority : INT;
	//Alarm delay setpoint(seconds)
	{attribute 'OPC.UA.DA' :='1'}
	popa_0081_cct_3142_a_high_delay_setpoint : INT;
	//Alarm active for HMI
	{attribute 'OPC.UA.DA' :='1'}
	popa_0081_cct_3142_a_high_active : BOOL;
	//Analog Alarm Setpoint
	{attribute 'OPC.UA.DA' :='1'}
	popa_0081_cct_3142_a_high_setpoint : REAL;
	//Alarm enable
	{attribute 'OPC.UA.DA' :='1'}
	popa_0081_cct_3142_a_high_enable: BOOL;
	
	//Alarm Priority setpoint
	{attribute 'OPC.UA.DA' :='1'}
	popa_0081_cct_3142_a_high_high_priority : INT;
	//Alarm delay setpoint(seconds)
	{attribute 'OPC.UA.DA' :='1'}
	popa_0081_cct_3142_a_high_high_delay_setpoint : INT;
	//Alarm active for HMI
	{attribute 'OPC.UA.DA' :='1'}
	popa_0081_cct_3142_a_high_high_active : BOOL;
	//Analog Alarm Setpoint
	{attribute 'OPC.UA.DA' :='1'}
	popa_0081_cct_3142_a_high_high_setpoint : REAL;
	//Alarm enable
	{attribute 'OPC.UA.DA' :='1'}
	popa_0081_cct_3142_a_high_high_enable: BOOL;
	
	
	//Raw Min value for analog input
	{attribute 'OPC.UA.DA' :='1'}
	popa_0081_cct_3142_a_raw_min : REAL :=0;
	//Raw max value for analog input
	{attribute 'OPC.UA.DA' :='1'}
	popa_0081_cct_3142_a_raw_max : REAL :=32767;
	//EU Min value for analog input
	{attribute 'OPC.UA.DA' :='1'}
	popa_0081_cct_3142_a_eu_min : REAL;
	//EU Max value for analog input
	{attribute 'OPC.UA.DA' :='1'}
	popa_0081_cct_3142_a_eu_max : REAL;
	//Filter factor value for analog input
	{attribute 'OPC.UA.DA' :='1'}
	popa_0081_cct_3142_a_filter_factor : REAL;
	//Scaled value for analog input
	{attribute 'OPC.UA.DA' :='1'}
	popa_0081_cct_3142_a_scaled_value : REAL;
	
		//---cct_3242-----------------------------------------------------------------------------------------------------------------------
	//Alarm Priority setpoint
	{attribute 'OPC.UA.DA' :='1'}
	popa_0081_cct_3242_a_low_low_priority : INT;
	//Alarm delay setpoint(seconds)
	{attribute 'OPC.UA.DA' :='1'}
	popa_0081_cct_3242_a_low_low_delay_setpoint : INT;
	//Alarm active for HMI
	{attribute 'OPC.UA.DA' :='1'}
	popa_0081_cct_3242_a_low_low_active : BOOL;
	//Analog Alarm Setpoint
	{attribute 'OPC.UA.DA' :='1'}
	popa_0081_cct_3242_a_low_low_setpoint : REAL;
	//Alarm enable
	{attribute 'OPC.UA.DA' :='1'}
	popa_0081_cct_3242_a_low_low_enable: BOOL;
	
	//Alarm Priority setpoint
	{attribute 'OPC.UA.DA' :='1'}
	popa_0081_cct_3242_a_low_priority : INT;
	//Alarm delay setpoint(seconds)
	{attribute 'OPC.UA.DA' :='1'}
	popa_0081_cct_3242_a_low_delay_setpoint : INT;
	//Alarm active for HMI
	{attribute 'OPC.UA.DA' :='1'}
	popa_0081_cct_3242_a_low_active : BOOL;
	//Analog Alarm Setpoint
	{attribute 'OPC.UA.DA' :='1'}
	popa_0081_cct_3242_a_low_setpoint : REAL;
	//Alarm enable
	{attribute 'OPC.UA.DA' :='1'}
	popa_0081_cct_3242_a_low_enable: BOOL;
	
	//Alarm Priority setpoint
	{attribute 'OPC.UA.DA' :='1'}
	popa_0081_cct_3242_a_high_priority : INT;
	//Alarm delay setpoint(seconds)
	{attribute 'OPC.UA.DA' :='1'}
	popa_0081_cct_3242_a_high_delay_setpoint : INT;
	//Alarm active for HMI
	{attribute 'OPC.UA.DA' :='1'}
	popa_0081_cct_3242_a_high_active : BOOL;
	//Analog Alarm Setpoint
	{attribute 'OPC.UA.DA' :='1'}
	popa_0081_cct_3242_a_high_setpoint : REAL;
	//Alarm enable
	{attribute 'OPC.UA.DA' :='1'}
	popa_0081_cct_3242_a_high_enable: BOOL;
	
	//Alarm Priority setpoint
	{attribute 'OPC.UA.DA' :='1'}
	popa_0081_cct_3242_a_high_high_priority : INT;
	//Alarm delay setpoint(seconds)
	{attribute 'OPC.UA.DA' :='1'}
	popa_0081_cct_3242_a_high_high_delay_setpoint : INT;
	//Alarm active for HMI
	{attribute 'OPC.UA.DA' :='1'}
	popa_0081_cct_3242_a_high_high_active : BOOL;
	//Analog Alarm Setpoint
	{attribute 'OPC.UA.DA' :='1'}
	popa_0081_cct_3242_a_high_high_setpoint : REAL;
	//Alarm enable
	{attribute 'OPC.UA.DA' :='1'}
	popa_0081_cct_3242_a_high_high_enable: BOOL;
	
	
	//Raw Min value for analog input
	{attribute 'OPC.UA.DA' :='1'}
	popa_0081_cct_3242_a_raw_min : REAL :=0;
	//Raw max value for analog input
	{attribute 'OPC.UA.DA' :='1'}
	popa_0081_cct_3242_a_raw_max : REAL :=32767;
	//EU Min value for analog input
	{attribute 'OPC.UA.DA' :='1'}
	popa_0081_cct_3242_a_eu_min : REAL;
	//EU Max value for analog input
	{attribute 'OPC.UA.DA' :='1'}
	popa_0081_cct_3242_a_eu_max : REAL;
	//Filter factor value for analog input
	{attribute 'OPC.UA.DA' :='1'}
	popa_0081_cct_3242_a_filter_factor : REAL;
	//Scaled value for analog input
	{attribute 'OPC.UA.DA' :='1'}
	popa_0081_cct_3242_a_scaled_value : REAL;
	
		//---cct_3342-----------------------------------------------------------------------------------------------------------------------
	//Alarm Priority setpoint
	{attribute 'OPC.UA.DA' :='1'}
	popa_0081_cct_3342_a_low_low_priority : INT;
	//Alarm delay setpoint(seconds)
	{attribute 'OPC.UA.DA' :='1'}
	popa_0081_cct_3342_a_low_low_delay_setpoint : INT;
	//Alarm active for HMI
	{attribute 'OPC.UA.DA' :='1'}
	popa_0081_cct_3342_a_low_low_active : BOOL;
	//Analog Alarm Setpoint
	{attribute 'OPC.UA.DA' :='1'}
	popa_0081_cct_3342_a_low_low_setpoint : REAL;
	//Alarm enable
	{attribute 'OPC.UA.DA' :='1'}
	popa_0081_cct_3342_a_low_low_enable: BOOL;
	
	//Alarm Priority setpoint
	{attribute 'OPC.UA.DA' :='1'}
	popa_0081_cct_3342_a_low_priority : INT;
	//Alarm delay setpoint(seconds)
	{attribute 'OPC.UA.DA' :='1'}
	popa_0081_cct_3342_a_low_delay_setpoint : INT;
	//Alarm active for HMI
	{attribute 'OPC.UA.DA' :='1'}
	popa_0081_cct_3342_a_low_active : BOOL;
	//Analog Alarm Setpoint
	{attribute 'OPC.UA.DA' :='1'}
	popa_0081_cct_3342_a_low_setpoint : REAL;
	//Alarm enable
	{attribute 'OPC.UA.DA' :='1'}
	popa_0081_cct_3342_a_low_enable: BOOL;
	
	//Alarm Priority setpoint
	{attribute 'OPC.UA.DA' :='1'}
	popa_0081_cct_3342_a_high_priority : INT;
	//Alarm delay setpoint(seconds)
	{attribute 'OPC.UA.DA' :='1'}
	popa_0081_cct_3342_a_high_delay_setpoint : INT;
	//Alarm active for HMI
	{attribute 'OPC.UA.DA' :='1'}
	popa_0081_cct_3342_a_high_active : BOOL;
	//Analog Alarm Setpoint
	{attribute 'OPC.UA.DA' :='1'}
	popa_0081_cct_3342_a_high_setpoint : REAL;
	//Alarm enable
	{attribute 'OPC.UA.DA' :='1'}
	popa_0081_cct_3342_a_high_enable: BOOL;
	
	//Alarm Priority setpoint
	{attribute 'OPC.UA.DA' :='1'}
	popa_0081_cct_3342_a_high_high_priority : INT;
	//Alarm delay setpoint(seconds)
	{attribute 'OPC.UA.DA' :='1'}
	popa_0081_cct_3342_a_high_high_delay_setpoint : INT;
	//Alarm active for HMI
	{attribute 'OPC.UA.DA' :='1'}
	popa_0081_cct_3342_a_high_high_active : BOOL;
	//Analog Alarm Setpoint
	{attribute 'OPC.UA.DA' :='1'}
	popa_0081_cct_3342_a_high_high_setpoint : REAL;
	//Alarm enable
	{attribute 'OPC.UA.DA' :='1'}
	popa_0081_cct_3342_a_high_high_enable: BOOL;
	
	
	//Raw Min value for analog input
	{attribute 'OPC.UA.DA' :='1'}
	popa_0081_cct_3342_a_raw_min : REAL :=0;
	//Raw max value for analog input
	{attribute 'OPC.UA.DA' :='1'}
	popa_0081_cct_3342_a_raw_max : REAL :=32767;
	//EU Min value for analog input
	{attribute 'OPC.UA.DA' :='1'}
	popa_0081_cct_3342_a_eu_min : REAL;
	//EU Max value for analog input
	{attribute 'OPC.UA.DA' :='1'}
	popa_0081_cct_3342_a_eu_max : REAL;
	//Filter factor value for analog input
	{attribute 'OPC.UA.DA' :='1'}
	popa_0081_cct_3342_a_filter_factor : REAL;
	//Scaled value for analog input
	{attribute 'OPC.UA.DA' :='1'}
	popa_0081_cct_3342_a_scaled_value : REAL;

	//---ft_3122-----------------------------------------------------------------------------------------------------------------------
	//Alarm Priority setpoint
	{attribute 'OPC.UA.DA' :='1'}
	popa_0081_ft_3122_a_low_low_priority : INT;
	//Alarm delay setpoint(seconds)
	{attribute 'OPC.UA.DA' :='1'}
	popa_0081_ft_3122_a_low_low_delay_setpoint : INT;
	//Alarm active for HMI
	{attribute 'OPC.UA.DA' :='1'}
	popa_0081_ft_3122_a_low_low_active : BOOL;
	//Analog Alarm Setpoint
	{attribute 'OPC.UA.DA' :='1'}
	popa_0081_ft_3122_a_low_low_setpoint : REAL;
	//Alarm enable
	{attribute 'OPC.UA.DA' :='1'}
	popa_0081_ft_3122_a_low_low_enable: BOOL;
	
	//Alarm Priority setpoint
	{attribute 'OPC.UA.DA' :='1'}
	popa_0081_ft_3122_a_low_priority : INT;
	//Alarm delay setpoint(seconds)
	{attribute 'OPC.UA.DA' :='1'}
	popa_0081_ft_3122_a_low_delay_setpoint : INT;
	//Alarm active for HMI
	{attribute 'OPC.UA.DA' :='1'}
	popa_0081_ft_3122_a_low_active : BOOL;
	//Analog Alarm Setpoint
	{attribute 'OPC.UA.DA' :='1'}
	popa_0081_ft_3122_a_low_setpoint : REAL;
	//Alarm enable
	{attribute 'OPC.UA.DA' :='1'}
	popa_0081_ft_3122_a_low_enable: BOOL;
	
	//Alarm Priority setpoint
	{attribute 'OPC.UA.DA' :='1'}
	popa_0081_ft_3122_a_high_priority : INT;
	//Alarm delay setpoint(seconds)
	{attribute 'OPC.UA.DA' :='1'}
	popa_0081_ft_3122_a_high_delay_setpoint : INT;
	//Alarm active for HMI
	{attribute 'OPC.UA.DA' :='1'}
	popa_0081_ft_3122_a_high_active : BOOL;
	//Analog Alarm Setpoint
	{attribute 'OPC.UA.DA' :='1'}
	popa_0081_ft_3122_a_high_setpoint : REAL;
	//Alarm enable
	{attribute 'OPC.UA.DA' :='1'}
	popa_0081_ft_3122_a_high_enable: BOOL;
	
	//Alarm Priority setpoint
	{attribute 'OPC.UA.DA' :='1'}
	popa_0081_ft_3122_a_high_high_priority : INT;
	//Alarm delay setpoint(seconds)
	{attribute 'OPC.UA.DA' :='1'}
	popa_0081_ft_3122_a_high_high_delay_setpoint : INT;
	//Alarm active for HMI
	{attribute 'OPC.UA.DA' :='1'}
	popa_0081_ft_3122_a_high_high_active : BOOL;
	//Analog Alarm Setpoint
	{attribute 'OPC.UA.DA' :='1'}
	popa_0081_ft_3122_a_high_high_setpoint : REAL;
	//Alarm enable
	{attribute 'OPC.UA.DA' :='1'}
	popa_0081_ft_3122_a_high_high_enable: BOOL;
	
	
	//Raw Min value for analog input
	{attribute 'OPC.UA.DA' :='1'}
	popa_0081_ft_3122_a_raw_min : REAL :=0;
	//Raw max value for analog input
	{attribute 'OPC.UA.DA' :='1'}
	popa_0081_ft_3122_a_raw_max : REAL :=32767;
	//EU Min value for analog input
	{attribute 'OPC.UA.DA' :='1'}
	popa_0081_ft_3122_a_eu_min : REAL;
	//EU Max value for analog input
	{attribute 'OPC.UA.DA' :='1'}
	popa_0081_ft_3122_a_eu_max : REAL;
	//Filter factor value for analog input
	{attribute 'OPC.UA.DA' :='1'}
	popa_0081_ft_3122_a_filter_factor : REAL;
	//Scaled value for analog input
	{attribute 'OPC.UA.DA' :='1'}
	popa_0081_ft_3122_a_scaled_value : REAL;
	
	//---ft_3222-----------------------------------------------------------------------------------------------------------------------
	//Alarm Priority setpoint
	{attribute 'OPC.UA.DA' :='1'}
	popa_0081_ft_3222_a_low_low_priority : INT;
	//Alarm delay setpoint(seconds)
	{attribute 'OPC.UA.DA' :='1'}
	popa_0081_ft_3222_a_low_low_delay_setpoint : INT;
	//Alarm active for HMI
	{attribute 'OPC.UA.DA' :='1'}
	popa_0081_ft_3222_a_low_low_active : BOOL;
	//Analog Alarm Setpoint
	{attribute 'OPC.UA.DA' :='1'}
	popa_0081_ft_3222_a_low_low_setpoint : REAL;
	//Alarm enable
	{attribute 'OPC.UA.DA' :='1'}
	popa_0081_ft_3222_a_low_low_enable: BOOL;
	
	//Alarm Priority setpoint
	{attribute 'OPC.UA.DA' :='1'}
	popa_0081_ft_3222_a_low_priority : INT;
	//Alarm delay setpoint(seconds)
	{attribute 'OPC.UA.DA' :='1'}
	popa_0081_ft_3222_a_low_delay_setpoint : INT;
	//Alarm active for HMI
	{attribute 'OPC.UA.DA' :='1'}
	popa_0081_ft_3222_a_low_active : BOOL;
	//Analog Alarm Setpoint
	{attribute 'OPC.UA.DA' :='1'}
	popa_0081_ft_3222_a_low_setpoint : REAL;
	//Alarm enable
	{attribute 'OPC.UA.DA' :='1'}
	popa_0081_ft_3222_a_low_enable: BOOL;
	
	//Alarm Priority setpoint
	{attribute 'OPC.UA.DA' :='1'}
	popa_0081_ft_3222_a_high_priority : INT;
	//Alarm delay setpoint(seconds)
	{attribute 'OPC.UA.DA' :='1'}
	popa_0081_ft_3222_a_high_delay_setpoint : INT;
	//Alarm active for HMI
	{attribute 'OPC.UA.DA' :='1'}
	popa_0081_ft_3222_a_high_active : BOOL;
	//Analog Alarm Setpoint
	{attribute 'OPC.UA.DA' :='1'}
	popa_0081_ft_3222_a_high_setpoint : REAL;
	//Alarm enable
	{attribute 'OPC.UA.DA' :='1'}
	popa_0081_ft_3222_a_high_enable: BOOL;
	
	//Alarm Priority setpoint
	{attribute 'OPC.UA.DA' :='1'}
	popa_0081_ft_3222_a_high_high_priority : INT;
	//Alarm delay setpoint(seconds)
	{attribute 'OPC.UA.DA' :='1'}
	popa_0081_ft_3222_a_high_high_delay_setpoint : INT;
	//Alarm active for HMI
	{attribute 'OPC.UA.DA' :='1'}
	popa_0081_ft_3222_a_high_high_active : BOOL;
	//Analog Alarm Setpoint
	{attribute 'OPC.UA.DA' :='1'}
	popa_0081_ft_3222_a_high_high_setpoint : REAL;
	//Alarm enable
	{attribute 'OPC.UA.DA' :='1'}
	popa_0081_ft_3222_a_high_high_enable: BOOL;
	
	
	//Raw Min value for analog input
	{attribute 'OPC.UA.DA' :='1'}
	popa_0081_ft_3222_a_raw_min : REAL :=0;
	//Raw max value for analog input
	{attribute 'OPC.UA.DA' :='1'}
	popa_0081_ft_3222_a_raw_max : REAL :=32767;
	//EU Min value for analog input
	{attribute 'OPC.UA.DA' :='1'}
	popa_0081_ft_3222_a_eu_min : REAL;
	//EU Max value for analog input
	{attribute 'OPC.UA.DA' :='1'}
	popa_0081_ft_3222_a_eu_max : REAL;
	//Filter factor value for analog input
	{attribute 'OPC.UA.DA' :='1'}
	popa_0081_ft_3222_a_filter_factor : REAL;
	//Scaled value for analog input
	{attribute 'OPC.UA.DA' :='1'}
	popa_0081_ft_3222_a_scaled_value : REAL;
	
	//---ft_3322-----------------------------------------------------------------------------------------------------------------------
	//Alarm Priority setpoint
	{attribute 'OPC.UA.DA' :='1'}
	popa_0081_ft_3322_a_low_low_priority : INT;
	//Alarm delay setpoint(seconds)
	{attribute 'OPC.UA.DA' :='1'}
	popa_0081_ft_3322_a_low_low_delay_setpoint : INT;
	//Alarm active for HMI
	{attribute 'OPC.UA.DA' :='1'}
	popa_0081_ft_3322_a_low_low_active : BOOL;
	//Analog Alarm Setpoint
	{attribute 'OPC.UA.DA' :='1'}
	popa_0081_ft_3322_a_low_low_setpoint : REAL;
	//Alarm enable
	{attribute 'OPC.UA.DA' :='1'}
	popa_0081_ft_3322_a_low_low_enable: BOOL;
	
	//Alarm Priority setpoint
	{attribute 'OPC.UA.DA' :='1'}
	popa_0081_ft_3322_a_low_priority : INT;
	//Alarm delay setpoint(seconds)
	{attribute 'OPC.UA.DA' :='1'}
	popa_0081_ft_3322_a_low_delay_setpoint : INT;
	//Alarm active for HMI
	{attribute 'OPC.UA.DA' :='1'}
	popa_0081_ft_3322_a_low_active : BOOL;
	//Analog Alarm Setpoint
	{attribute 'OPC.UA.DA' :='1'}
	popa_0081_ft_3322_a_low_setpoint : REAL;
	//Alarm enable
	{attribute 'OPC.UA.DA' :='1'}
	popa_0081_ft_3322_a_low_enable: BOOL;
	
	//Alarm Priority setpoint
	{attribute 'OPC.UA.DA' :='1'}
	popa_0081_ft_3322_a_high_priority : INT;
	//Alarm delay setpoint(seconds)
	{attribute 'OPC.UA.DA' :='1'}
	popa_0081_ft_3322_a_high_delay_setpoint : INT;
	//Alarm active for HMI
	{attribute 'OPC.UA.DA' :='1'}
	popa_0081_ft_3322_a_high_active : BOOL;
	//Analog Alarm Setpoint
	{attribute 'OPC.UA.DA' :='1'}
	popa_0081_ft_3322_a_high_setpoint : REAL;
	//Alarm enable
	{attribute 'OPC.UA.DA' :='1'}
	popa_0081_ft_3322_a_high_enable: BOOL;
	
	//Alarm Priority setpoint
	{attribute 'OPC.UA.DA' :='1'}
	popa_0081_ft_3322_a_high_high_priority : INT;
	//Alarm delay setpoint(seconds)
	{attribute 'OPC.UA.DA' :='1'}
	popa_0081_ft_3322_a_high_high_delay_setpoint : INT;
	//Alarm active for HMI
	{attribute 'OPC.UA.DA' :='1'}
	popa_0081_ft_3322_a_high_high_active : BOOL;
	//Analog Alarm Setpoint
	{attribute 'OPC.UA.DA' :='1'}
	popa_0081_ft_3322_a_high_high_setpoint : REAL;
	//Alarm enable
	{attribute 'OPC.UA.DA' :='1'}
	popa_0081_ft_3322_a_high_high_enable: BOOL;
	
	
	//Raw Min value for analog input
	{attribute 'OPC.UA.DA' :='1'}
	popa_0081_ft_3322_a_raw_min : REAL :=0;
	//Raw max value for analog input
	{attribute 'OPC.UA.DA' :='1'}
	popa_0081_ft_3322_a_raw_max : REAL :=32767;
	//EU Min value for analog input
	{attribute 'OPC.UA.DA' :='1'}
	popa_0081_ft_3322_a_eu_min : REAL;
	//EU Max value for analog input
	{attribute 'OPC.UA.DA' :='1'}
	popa_0081_ft_3322_a_eu_max : REAL;
	//Filter factor value for analog input
	{attribute 'OPC.UA.DA' :='1'}
	popa_0081_ft_3322_a_filter_factor : REAL;
	//Scaled value for analog input
	{attribute 'OPC.UA.DA' :='1'}
	popa_0081_ft_3322_a_scaled_value : REAL;
	
	//---lt_3102-----------------------------------------------------------------------------------------------------------------------
	//Alarm Priority setpoint
	{attribute 'OPC.UA.DA' :='1'}
	popa_0081_lt_3102_a_low_low_priority : INT;
	//Alarm delay setpoint(seconds)
	{attribute 'OPC.UA.DA' :='1'}
	popa_0081_lt_3102_a_low_low_delay_setpoint : INT;
	//Alarm active for HMI
	{attribute 'OPC.UA.DA' :='1'}
	popa_0081_lt_3102_a_low_low_active : BOOL;
	//Analog Alarm Setpoint
	{attribute 'OPC.UA.DA' :='1'}
	popa_0081_lt_3102_a_low_low_setpoint : REAL;
	//Alarm enable
	{attribute 'OPC.UA.DA' :='1'}
	popa_0081_lt_3102_a_low_low_enable: BOOL;
	
	//Alarm Priority setpoint
	{attribute 'OPC.UA.DA' :='1'}
	popa_0081_lt_3102_a_low_priority : INT;
	//Alarm delay setpoint(seconds)
	{attribute 'OPC.UA.DA' :='1'}
	popa_0081_lt_3102_a_low_delay_setpoint : INT;
	//Alarm active for HMI
	{attribute 'OPC.UA.DA' :='1'}
	popa_0081_lt_3102_a_low_active : BOOL;
	//Analog Alarm Setpoint
	{attribute 'OPC.UA.DA' :='1'}
	popa_0081_lt_3102_a_low_setpoint : REAL;
	//Alarm enable
	{attribute 'OPC.UA.DA' :='1'}
	popa_0081_lt_3102_a_low_enable: BOOL;
	
	//Alarm Priority setpoint
	{attribute 'OPC.UA.DA' :='1'}
	popa_0081_lt_3102_a_high_priority : INT;
	//Alarm delay setpoint(seconds)
	{attribute 'OPC.UA.DA' :='1'}
	popa_0081_lt_3102_a_high_delay_setpoint : INT;
	//Alarm active for HMI
	{attribute 'OPC.UA.DA' :='1'}
	popa_0081_lt_3102_a_high_active : BOOL;
	//Analog Alarm Setpoint
	{attribute 'OPC.UA.DA' :='1'}
	popa_0081_lt_3102_a_high_setpoint : REAL;
	//Alarm enable
	{attribute 'OPC.UA.DA' :='1'}
	popa_0081_lt_3102_a_high_enable: BOOL;
	
	//Alarm Priority setpoint
	{attribute 'OPC.UA.DA' :='1'}
	popa_0081_lt_3102_a_high_high_priority : INT;
	//Alarm delay setpoint(seconds)
	{attribute 'OPC.UA.DA' :='1'}
	popa_0081_lt_3102_a_high_high_delay_setpoint : INT;
	//Alarm active for HMI
	{attribute 'OPC.UA.DA' :='1'}
	popa_0081_lt_3102_a_high_high_active : BOOL;
	//Analog Alarm Setpoint
	{attribute 'OPC.UA.DA' :='1'}
	popa_0081_lt_3102_a_high_high_setpoint : REAL;
	//Alarm enable
	{attribute 'OPC.UA.DA' :='1'}
	popa_0081_lt_3102_a_high_high_enable: BOOL;
	
	
	//Raw Min value for analog input
	{attribute 'OPC.UA.DA' :='1'}
	popa_0081_lt_3102_a_raw_min : REAL :=0;
	//Raw max value for analog input
	{attribute 'OPC.UA.DA' :='1'}
	popa_0081_lt_3102_a_raw_max : REAL :=32767;
	//EU Min value for analog input
	{attribute 'OPC.UA.DA' :='1'}
	popa_0081_lt_3102_a_eu_min : REAL;
	//EU Max value for analog input
	{attribute 'OPC.UA.DA' :='1'}
	popa_0081_lt_3102_a_eu_max : REAL;
	//Filter factor value for analog input
	{attribute 'OPC.UA.DA' :='1'}
	popa_0081_lt_3102_a_filter_factor : REAL;
	//Scaled value for analog input
	{attribute 'OPC.UA.DA' :='1'}
	popa_0081_lt_3102_a_scaled_value : REAL;
	
	//---lt_3202-----------------------------------------------------------------------------------------------------------------------
	//Alarm Priority setpoint
	{attribute 'OPC.UA.DA' :='1'}
	popa_0081_lt_3202_a_low_low_priority : INT;
	//Alarm delay setpoint(seconds)
	{attribute 'OPC.UA.DA' :='1'}
	popa_0081_lt_3202_a_low_low_delay_setpoint : INT;
	//Alarm active for HMI
	{attribute 'OPC.UA.DA' :='1'}
	popa_0081_lt_3202_a_low_low_active : BOOL;
	//Analog Alarm Setpoint
	{attribute 'OPC.UA.DA' :='1'}
	popa_0081_lt_3202_a_low_low_setpoint : REAL;
	//Alarm enable
	{attribute 'OPC.UA.DA' :='1'}
	popa_0081_lt_3202_a_low_low_enable: BOOL;
	
	//Alarm Priority setpoint
	{attribute 'OPC.UA.DA' :='1'}
	popa_0081_lt_3202_a_low_priority : INT;
	//Alarm delay setpoint(seconds)
	{attribute 'OPC.UA.DA' :='1'}
	popa_0081_lt_3202_a_low_delay_setpoint : INT;
	//Alarm active for HMI
	{attribute 'OPC.UA.DA' :='1'}
	popa_0081_lt_3202_a_low_active : BOOL;
	//Analog Alarm Setpoint
	{attribute 'OPC.UA.DA' :='1'}
	popa_0081_lt_3202_a_low_setpoint : REAL;
	//Alarm enable
	{attribute 'OPC.UA.DA' :='1'}
	popa_0081_lt_3202_a_low_enable: BOOL;
	
	//Alarm Priority setpoint
	{attribute 'OPC.UA.DA' :='1'}
	popa_0081_lt_3202_a_high_priority : INT;
	//Alarm delay setpoint(seconds)
	{attribute 'OPC.UA.DA' :='1'}
	popa_0081_lt_3202_a_high_delay_setpoint : INT;
	//Alarm active for HMI
	{attribute 'OPC.UA.DA' :='1'}
	popa_0081_lt_3202_a_high_active : BOOL;
	//Analog Alarm Setpoint
	{attribute 'OPC.UA.DA' :='1'}
	popa_0081_lt_3202_a_high_setpoint : REAL;
	//Alarm enable
	{attribute 'OPC.UA.DA' :='1'}
	popa_0081_lt_3202_a_high_enable: BOOL;
	
